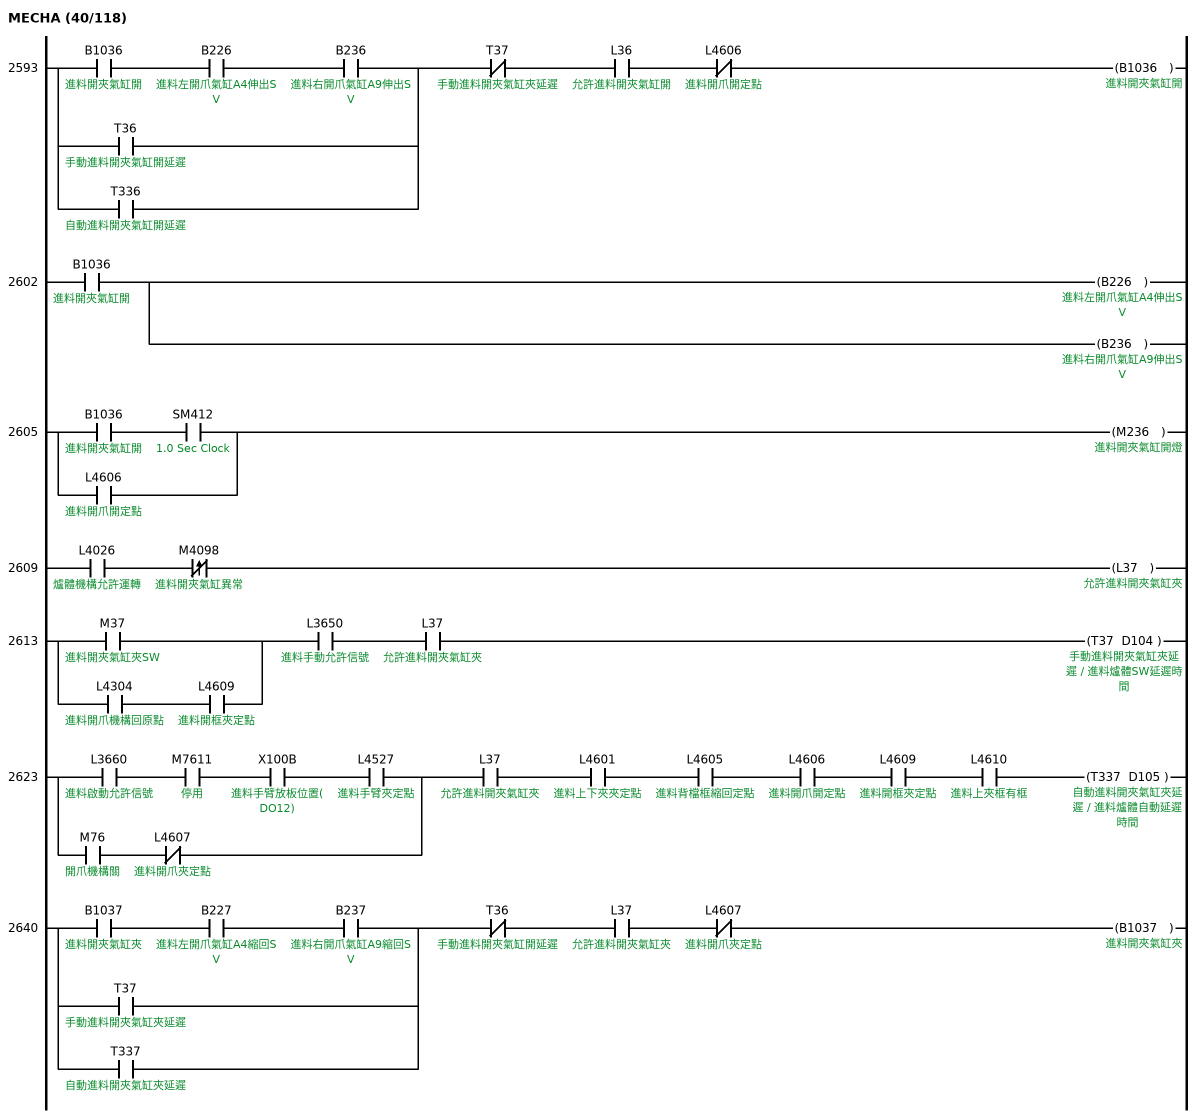
[picture p336: ladder of MECHA, rungs at steps 2593 to 2640]
2593  LD      B1036  ; 進料開夾氣缸開
      AND     B226  ; 進料左開爪氣缸A4伸出SV
      AND     B236  ; 進料右開爪氣缸A9伸出SV
      OR      T36  ; 手動進料開夾氣缸開延遲
      OR      T336  ; 自動進料開夾氣缸開延遲
      ANI     T37  ; 手動進料開夾氣缸夾延遲
      AND     L36  ; 允許進料開夾氣缸開
      ANI     L4606  ; 進料開爪開定點
      OUT     B1036  ; 進料開夾氣缸開
2602  LD      B1036  ; 進料開夾氣缸開
      OUT     B226  ; 進料左開爪氣缸A4伸出SV
      OUT     B236  ; 進料右開爪氣缸A9伸出SV
2605  LD      B1036  ; 進料開夾氣缸開
      AND     SM412  ; 1.0 Sec Clock
      OR      L4606  ; 進料開爪開定點
      OUT     M236  ; 進料開夾氣缸開燈
2609  LD      L4026  ; 爐體機構允許運轉
      ANDPI   M4098  ; 進料開夾氣缸異常
      OUT     L37  ; 允許進料開夾氣缸夾
2613  LD      M37  ; 進料開夾氣缸夾SW
      LD      L4304  ; 進料開爪機構回原點
      AND     L4609  ; 進料開框夾定點
      ORB
      AND     L3650  ; 進料手動允許信號
      AND     L37  ; 允許進料開夾氣缸夾
      OUT     T37 D104  ; 手動進料開夾氣缸夾延遲 / 進料爐體SW延遲時間
2623  LD      L3660  ; 進料啟動允許信號
      AND     M7611  ; 停用
      AND     X100B  ; 進料手臂放板位置(DO12)
      AND     L4527  ; 進料手臂夾定點
      LD      M76  ; 開爪機構關
      ANI     L4607  ; 進料開爪夾定點
      ORB
      AND     L37  ; 允許進料開夾氣缸夾
      AND     L4601  ; 進料上下夾夾定點
      AND     L4605  ; 進料背檔框縮回定點
      AND     L4606  ; 進料開爪開定點
      AND     L4609  ; 進料開框夾定點
      AND     L4610  ; 進料上夾框有框
      OUT     T337 D105  ; 自動進料開夾氣缸夾延遲 / 進料爐體自動延遲時間
2640  LD      B1037  ; 進料開夾氣缸夾
      AND     B227  ; 進料左開爪氣缸A4縮回SV
      AND     B237  ; 進料右開爪氣缸A9縮回SV
      OR      T37  ; 手動進料開夾氣缸夾延遲
      OR      T337  ; 自動進料開夾氣缸夾延遲
      ANI     T36  ; 手動進料開夾氣缸開延遲
      AND     L37  ; 允許進料開夾氣缸夾
      ANI     L4607  ; 進料開爪夾定點
      OUT     B1037  ; 進料開夾氣缸夾
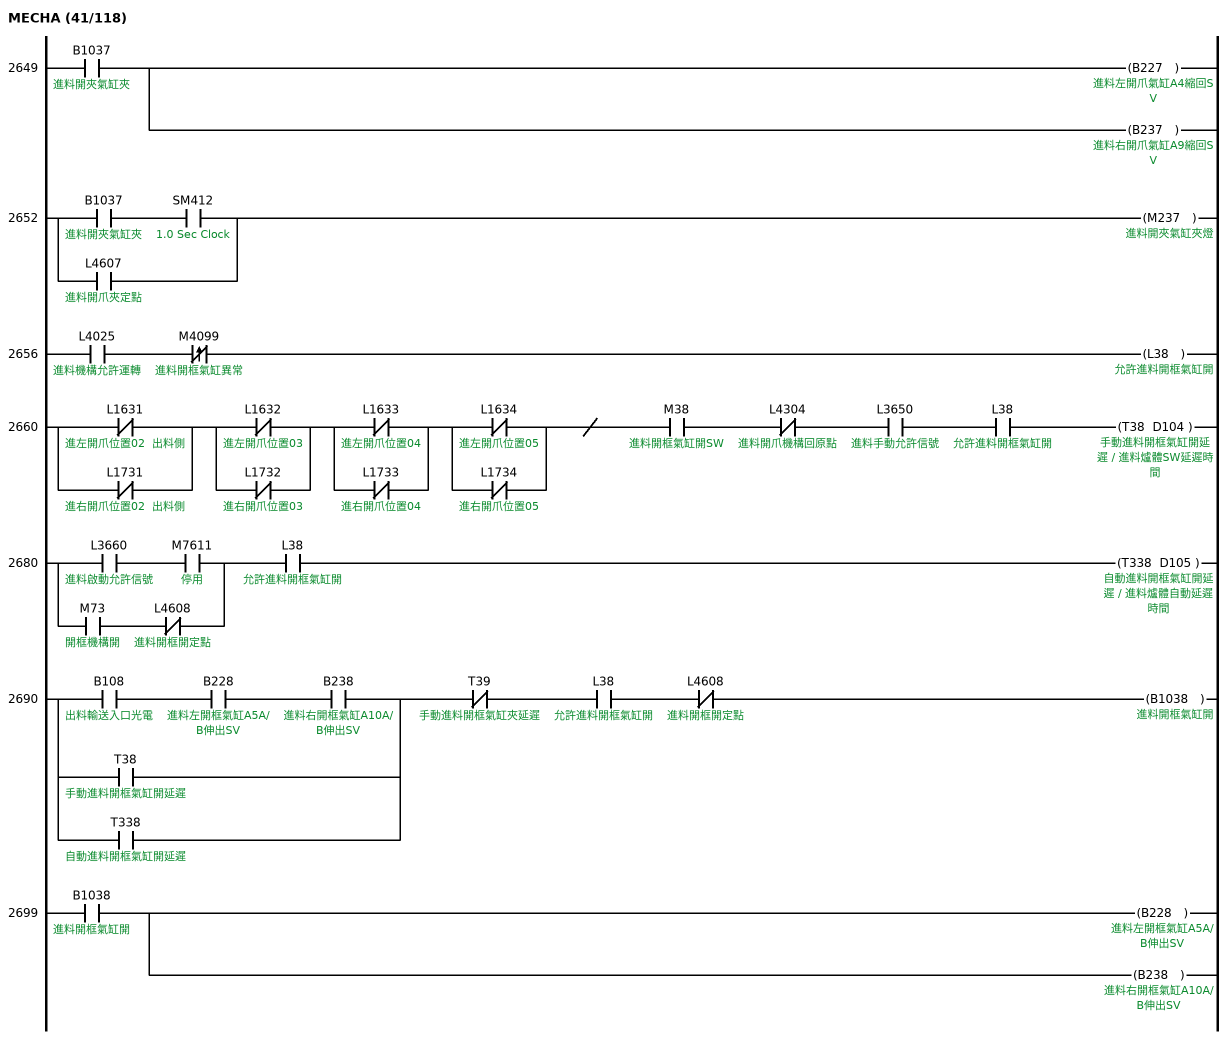
2649  LD      B1037  ; 進料開夾氣缸夾
      OUT     B227  ; 進料左開爪氣缸A4縮回SV
      OUT     B237  ; 進料右開爪氣缸A9縮回SV
2652  LD      B1037  ; 進料開夾氣缸夾
      AND     SM412  ; 1.0 Sec Clock
      OR      L4607  ; 進料開爪夾定點
      OUT     M237  ; 進料開夾氣缸夾燈
2656  LD      L4025  ; 進料機構允許運轉
      ANDPI   M4099  ; 進料開框氣缸異常
      OUT     L38  ; 允許進料開框氣缸開
2660  LDI     L1631  ; 進左開爪位置02  出料側
      ORI     L1731  ; 進右開爪位置02  出料側
      LDI     L1632  ; 進左開爪位置03
      ORI     L1732  ; 進右開爪位置03
      ANB
      LDI     L1633  ; 進左開爪位置04
      ORI     L1733  ; 進右開爪位置04
      ANB
      LDI     L1634  ; 進左開爪位置05
      ORI     L1734  ; 進右開爪位置05
      ANB
      INV
      AND     M38  ; 進料開框氣缸開SW
      ANI     L4304  ; 進料開爪機構回原點
      AND     L3650  ; 進料手動允許信號
      AND     L38  ; 允許進料開框氣缸開
      OUT     T38 D104  ; 手動進料開框氣缸開延遲 / 進料爐體SW延遲時間
2680  LD      L3660  ; 進料啟動允許信號
      AND     M7611  ; 停用
      LD      M73  ; 開框機構開
      ANI     L4608  ; 進料開框開定點
      ORB
      AND     L38  ; 允許進料開框氣缸開
      OUT     T338 D105  ; 自動進料開框氣缸開延遲 / 進料爐體自動延遲時間
2690  LD      B108  ; 出料輸送入口光電
      AND     B228  ; 進料左開框氣缸A5A/B伸出SV
      AND     B238  ; 進料右開框氣缸A10A/B伸出SV
      OR      T38  ; 手動進料開框氣缸開延遲
      OR      T338  ; 自動進料開框氣缸開延遲
      ANI     T39  ; 手動進料開框氣缸夾延遲
      AND     L38  ; 允許進料開框氣缸開
      ANI     L4608  ; 進料開框開定點
      OUT     B1038  ; 進料開框氣缸開
2699  LD      B1038  ; 進料開框氣缸開
      OUT     B228  ; 進料左開框氣缸A5A/B伸出SV
      OUT     B238  ; 進料右開框氣缸A10A/B伸出SV
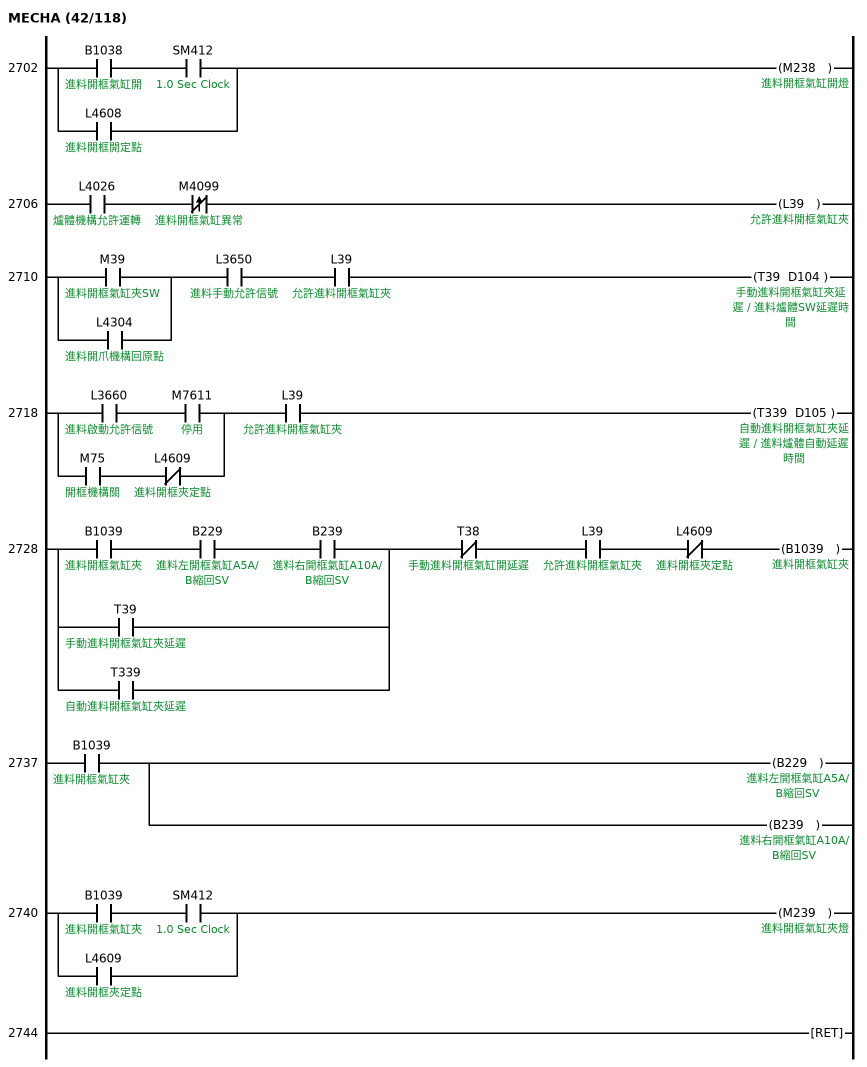
2702  LD      B1038  ; 進料開框氣缸開
      AND     SM412  ; 1.0 Sec Clock
      OR      L4608  ; 進料開框開定點
      OUT     M238  ; 進料開框氣缸開燈
2706  LD      L4026  ; 爐體機構允許運轉
      ANDPI   M4099  ; 進料開框氣缸異常
      OUT     L39  ; 允許進料開框氣缸夾
2710  LD      M39  ; 進料開框氣缸夾SW
      OR      L4304  ; 進料開爪機構回原點
      AND     L3650  ; 進料手動允許信號
      AND     L39  ; 允許進料開框氣缸夾
      OUT     T39 D104  ; 手動進料開框氣缸夾延遲 / 進料爐體SW延遲時間
2718  LD      L3660  ; 進料啟動允許信號
      AND     M7611  ; 停用
      LD      M75  ; 開框機構關
      ANI     L4609  ; 進料開框夾定點
      ORB
      AND     L39  ; 允許進料開框氣缸夾
      OUT     T339 D105  ; 自動進料開框氣缸夾延遲 / 進料爐體自動延遲時間
2728  LD      B1039  ; 進料開框氣缸夾
      AND     B229  ; 進料左開框氣缸A5A/B縮回SV
      AND     B239  ; 進料右開框氣缸A10A/B縮回SV
      OR      T39  ; 手動進料開框氣缸夾延遲
      OR      T339  ; 自動進料開框氣缸夾延遲
      ANI     T38  ; 手動進料開框氣缸開延遲
      AND     L39  ; 允許進料開框氣缸夾
      ANI     L4609  ; 進料開框夾定點
      OUT     B1039  ; 進料開框氣缸夾
2737  LD      B1039  ; 進料開框氣缸夾
      OUT     B229  ; 進料左開框氣缸A5A/B縮回SV
      OUT     B239  ; 進料右開框氣缸A10A/B縮回SV
2740  LD      B1039  ; 進料開框氣缸夾
      AND     SM412  ; 1.0 Sec Clock
      OR      L4609  ; 進料開框夾定點
      OUT     M239  ; 進料開框氣缸夾燈
2744  RET
      P1021
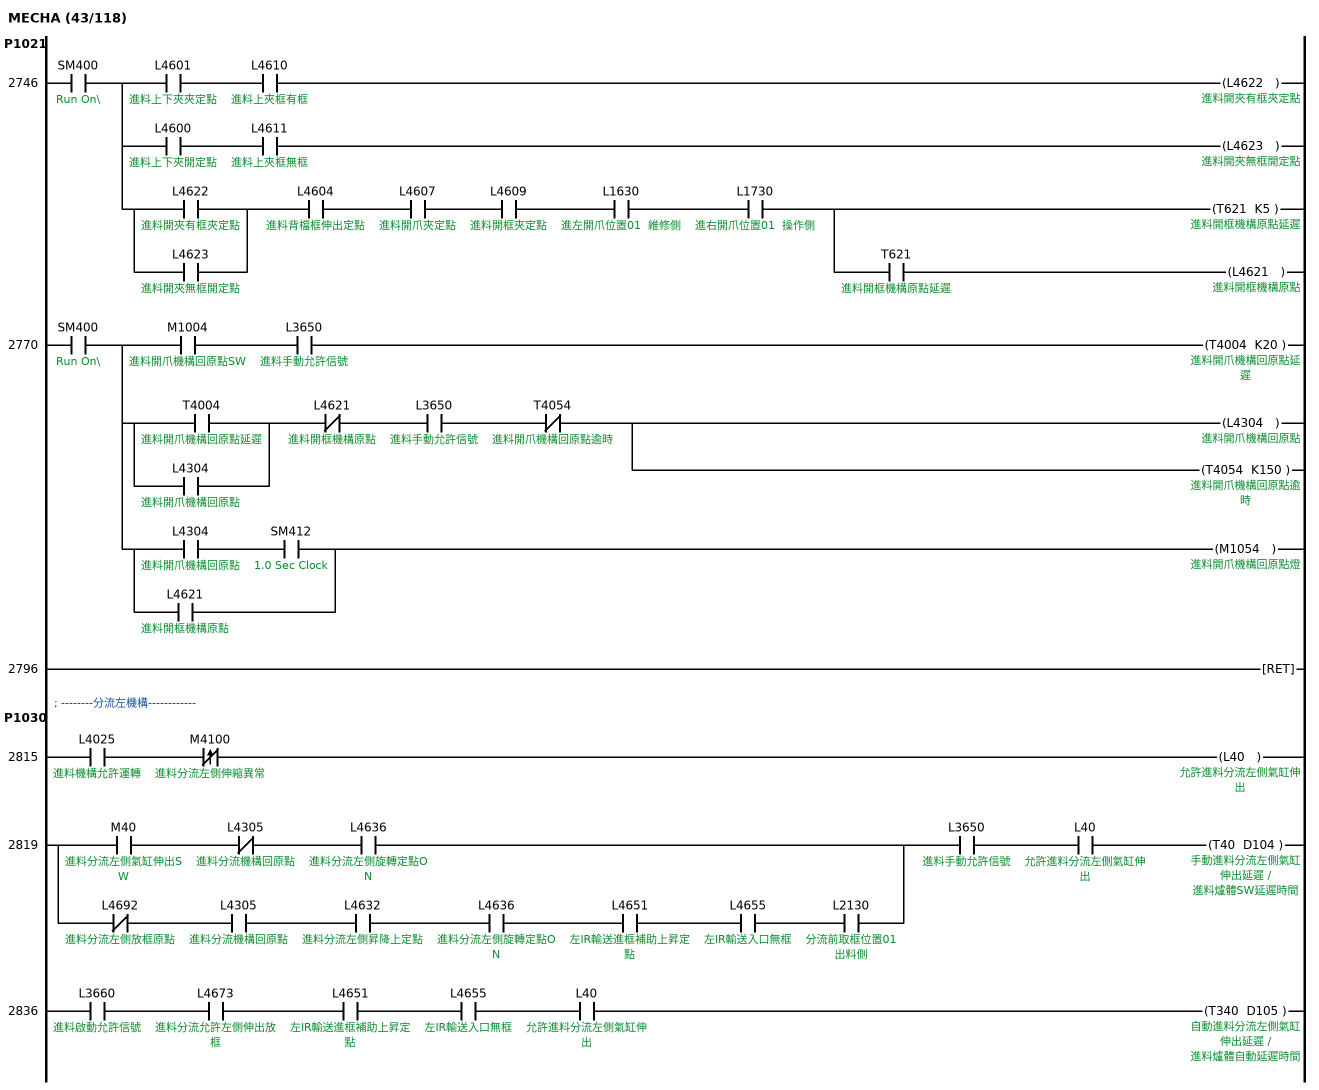
2746  LD      SM400  ; Run On\
      MPS
      AND     L4601  ; 進料上下夾夾定點
      AND     L4610  ; 進料上夾框有框
      OUT     L4622  ; 進料開夾有框夾定點
      MRD
      AND     L4600  ; 進料上下夾開定點
      AND     L4611  ; 進料上夾框無框
      OUT     L4623  ; 進料開夾無框開定點
      MPP
      LD      L4622  ; 進料開夾有框夾定點
      OR      L4623  ; 進料開夾無框開定點
      ANB
      AND     L4604  ; 進料背檔框伸出定點
      AND     L4607  ; 進料開爪夾定點
      AND     L4609  ; 進料開框夾定點
      AND     L1630  ; 進左開爪位置01  維修側
      AND     L1730  ; 進右開爪位置01  操作側
      OUT     T621 K5  ; 進料開框機構原點延遲
      AND     T621  ; 進料開框機構原點延遲
      OUT     L4621  ; 進料開框機構原點
2770  LD      SM400  ; Run On\
      MPS
      AND     M1004  ; 進料開爪機構回原點SW
      AND     L3650  ; 進料手動允許信號
      OUT     T4004 K20  ; 進料開爪機構回原點延遲
      MRD
      LD      T4004  ; 進料開爪機構回原點延遲
      OR      L4304  ; 進料開爪機構回原點
      ANB
      ANI     L4621  ; 進料開框機構原點
      AND     L3650  ; 進料手動允許信號
      ANI     T4054  ; 進料開爪機構回原點逾時
      OUT     L4304  ; 進料開爪機構回原點
      OUT     T4054 K150  ; 進料開爪機構回原點逾時
      MPP
      LD      L4304  ; 進料開爪機構回原點
      AND     SM412  ; 1.0 Sec Clock
      OR      L4621  ; 進料開框機構原點
      ANB
      OUT     M1054  ; 進料開爪機構回原點燈
2796  RET
; --------分流左機構------------
      P1030
2815  LD      L4025  ; 進料機構允許運轉
      ANDPI   M4100  ; 進料分流左側伸縮異常
      OUT     L40  ; 允許進料分流左側氣缸伸出
2819  LD      M40  ; 進料分流左側氣缸伸出SW
      ANI     L4305  ; 進料分流機構回原點
      AND     L4636  ; 進料分流左側旋轉定點ON
      LDI     L4692  ; 進料分流左側放框原點
      AND     L4305  ; 進料分流機構回原點
      AND     L4632  ; 進料分流左側昇降上定點
      AND     L4636  ; 進料分流左側旋轉定點ON
      AND     L4651  ; 左IR輸送進框補助上昇定點
      AND     L4655  ; 左IR輸送入口無框
      AND     L2130  ; 分流前取框位置01  出料側
      ORB
      AND     L3650  ; 進料手動允許信號
      AND     L40  ; 允許進料分流左側氣缸伸出
      OUT     T40 D104  ; 手動進料分流左側氣缸伸出延遲 / 進料爐體SW延遲時間
2836  LD      L3660  ; 進料啟動允許信號
      AND     L4673  ; 進料分流允許左側伸出放框
      AND     L4651  ; 左IR輸送進框補助上昇定點
      AND     L4655  ; 左IR輸送入口無框
      AND     L40  ; 允許進料分流左側氣缸伸出
      OUT     T340 D105  ; 自動進料分流左側氣缸伸出延遲 / 進料爐體自動延遲時間
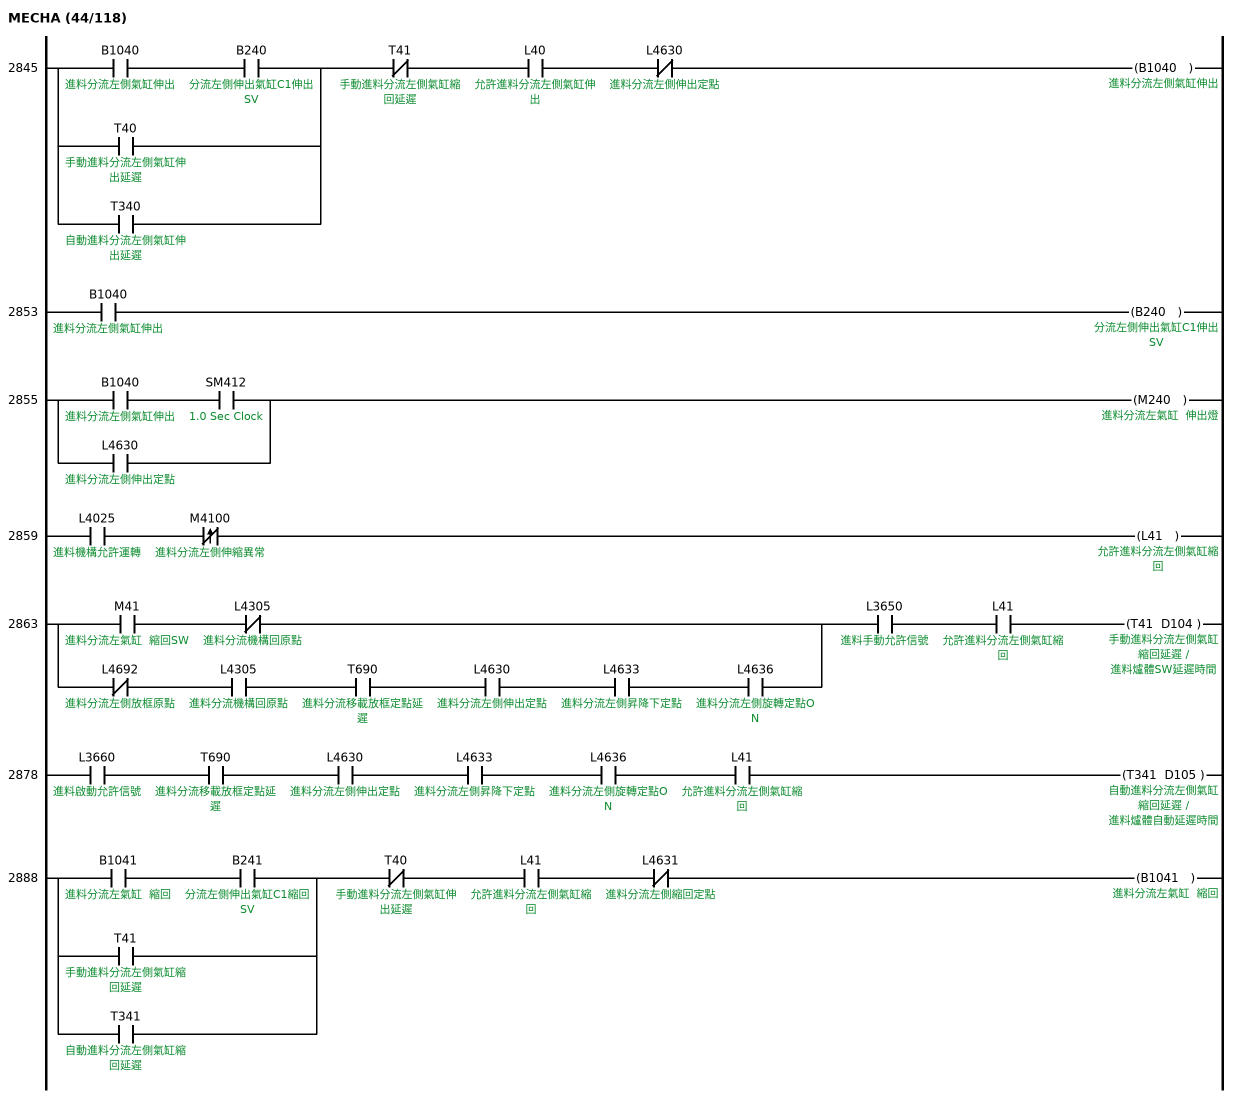
2845  LD      B1040  ; 進料分流左側氣缸伸出
      AND     B240  ; 分流左側伸出氣缸C1伸出SV
      OR      T40  ; 手動進料分流左側氣缸伸出延遲
      OR      T340  ; 自動進料分流左側氣缸伸出延遲
      ANI     T41  ; 手動進料分流左側氣缸縮回延遲
      AND     L40  ; 允許進料分流左側氣缸伸出
      ANI     L4630  ; 進料分流左側伸出定點
      OUT     B1040  ; 進料分流左側氣缸伸出
2853  LD      B1040  ; 進料分流左側氣缸伸出
      OUT     B240  ; 分流左側伸出氣缸C1伸出SV
2855  LD      B1040  ; 進料分流左側氣缸伸出
      AND     SM412  ; 1.0 Sec Clock
      OR      L4630  ; 進料分流左側伸出定點
      OUT     M240  ; 進料分流左氣缸  伸出燈
2859  LD      L4025  ; 進料機構允許運轉
      ANDPI   M4100  ; 進料分流左側伸縮異常
      OUT     L41  ; 允許進料分流左側氣缸縮回
2863  LD      M41  ; 進料分流左氣缸  縮回SW
      ANI     L4305  ; 進料分流機構回原點
      LDI     L4692  ; 進料分流左側放框原點
      AND     L4305  ; 進料分流機構回原點
      AND     T690  ; 進料分流移載放框定點延遲
      AND     L4630  ; 進料分流左側伸出定點
      AND     L4633  ; 進料分流左側昇降下定點
      AND     L4636  ; 進料分流左側旋轉定點ON
      ORB
      AND     L3650  ; 進料手動允許信號
      AND     L41  ; 允許進料分流左側氣缸縮回
      OUT     T41 D104  ; 手動進料分流左側氣缸縮回延遲 / 進料爐體SW延遲時間
2878  LD      L3660  ; 進料啟動允許信號
      AND     T690  ; 進料分流移載放框定點延遲
      AND     L4630  ; 進料分流左側伸出定點
      AND     L4633  ; 進料分流左側昇降下定點
      AND     L4636  ; 進料分流左側旋轉定點ON
      AND     L41  ; 允許進料分流左側氣缸縮回
      OUT     T341 D105  ; 自動進料分流左側氣缸縮回延遲 / 進料爐體自動延遲時間
2888  LD      B1041  ; 進料分流左氣缸  縮回
      AND     B241  ; 分流左側伸出氣缸C1縮回SV
      OR      T41  ; 手動進料分流左側氣缸縮回延遲
      OR      T341  ; 自動進料分流左側氣缸縮回延遲
      ANI     T40  ; 手動進料分流左側氣缸伸出延遲
      AND     L41  ; 允許進料分流左側氣缸縮回
      ANI     L4631  ; 進料分流左側縮回定點
      OUT     B1041  ; 進料分流左氣缸  縮回
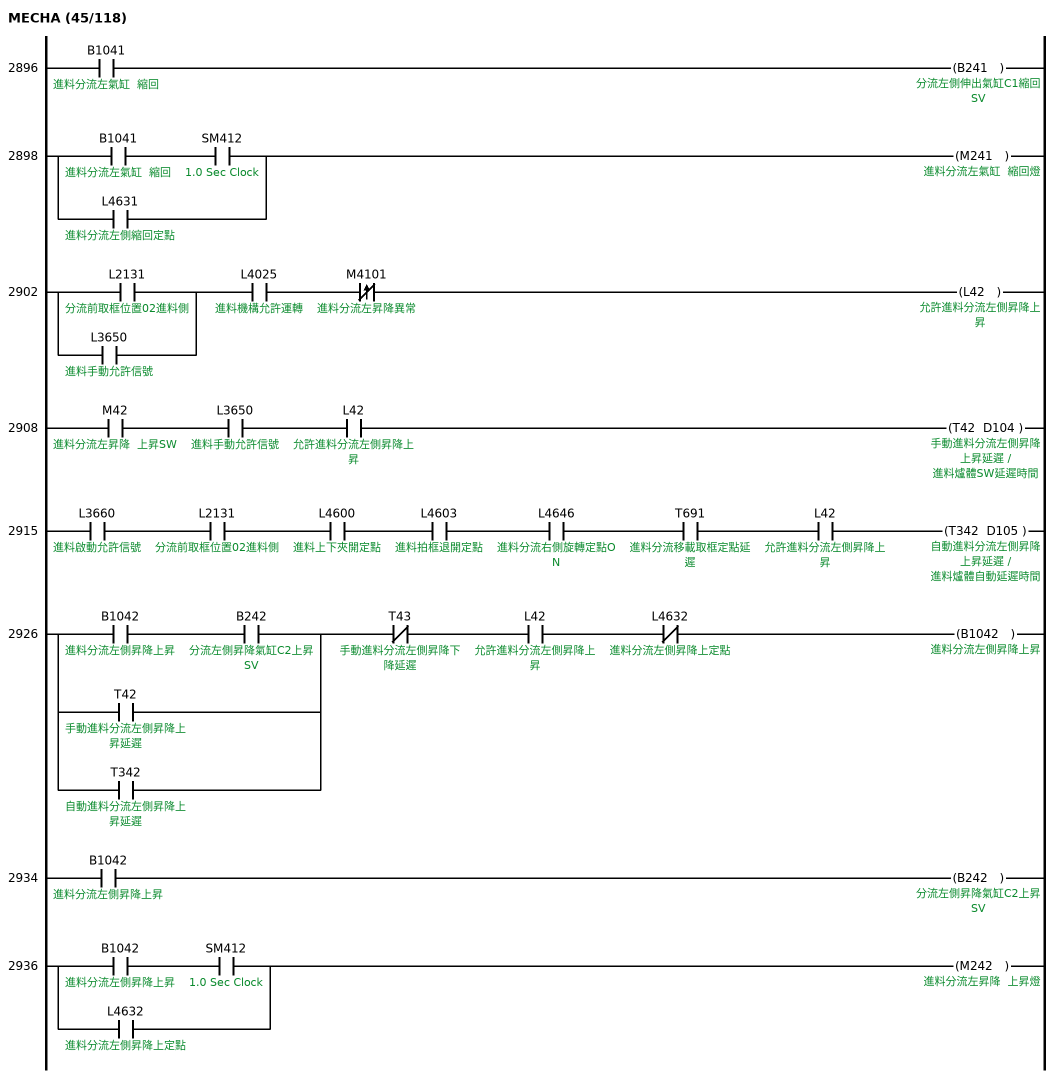
2896  LD      B1041  ; 進料分流左氣缸  縮回
      OUT     B241  ; 分流左側伸出氣缸C1縮回SV
2898  LD      B1041  ; 進料分流左氣缸  縮回
      AND     SM412  ; 1.0 Sec Clock
      OR      L4631  ; 進料分流左側縮回定點
      OUT     M241  ; 進料分流左氣缸  縮回燈
2902  LD      L2131  ; 分流前取框位置02進料側
      OR      L3650  ; 進料手動允許信號
      AND     L4025  ; 進料機構允許運轉
      ANDPI   M4101  ; 進料分流左昇降異常
      OUT     L42  ; 允許進料分流左側昇降上昇
2908  LD      M42  ; 進料分流左昇降  上昇SW
      AND     L3650  ; 進料手動允許信號
      AND     L42  ; 允許進料分流左側昇降上昇
      OUT     T42 D104  ; 手動進料分流左側昇降上昇延遲 / 進料爐體SW延遲時間
2915  LD      L3660  ; 進料啟動允許信號
      AND     L2131  ; 分流前取框位置02進料側
      AND     L4600  ; 進料上下夾開定點
      AND     L4603  ; 進料拍框退開定點
      AND     L4646  ; 進料分流右側旋轉定點ON
      AND     T691  ; 進料分流移載取框定點延遲
      AND     L42  ; 允許進料分流左側昇降上昇
      OUT     T342 D105  ; 自動進料分流左側昇降上昇延遲 / 進料爐體自動延遲時間
2926  LD      B1042  ; 進料分流左側昇降上昇
      AND     B242  ; 分流左側昇降氣缸C2上昇SV
      OR      T42  ; 手動進料分流左側昇降上昇延遲
      OR      T342  ; 自動進料分流左側昇降上昇延遲
      ANI     T43  ; 手動進料分流左側昇降下降延遲
      AND     L42  ; 允許進料分流左側昇降上昇
      ANI     L4632  ; 進料分流左側昇降上定點
      OUT     B1042  ; 進料分流左側昇降上昇
2934  LD      B1042  ; 進料分流左側昇降上昇
      OUT     B242  ; 分流左側昇降氣缸C2上昇SV
2936  LD      B1042  ; 進料分流左側昇降上昇
      AND     SM412  ; 1.0 Sec Clock
      OR      L4632  ; 進料分流左側昇降上定點
      OUT     M242  ; 進料分流左昇降  上昇燈
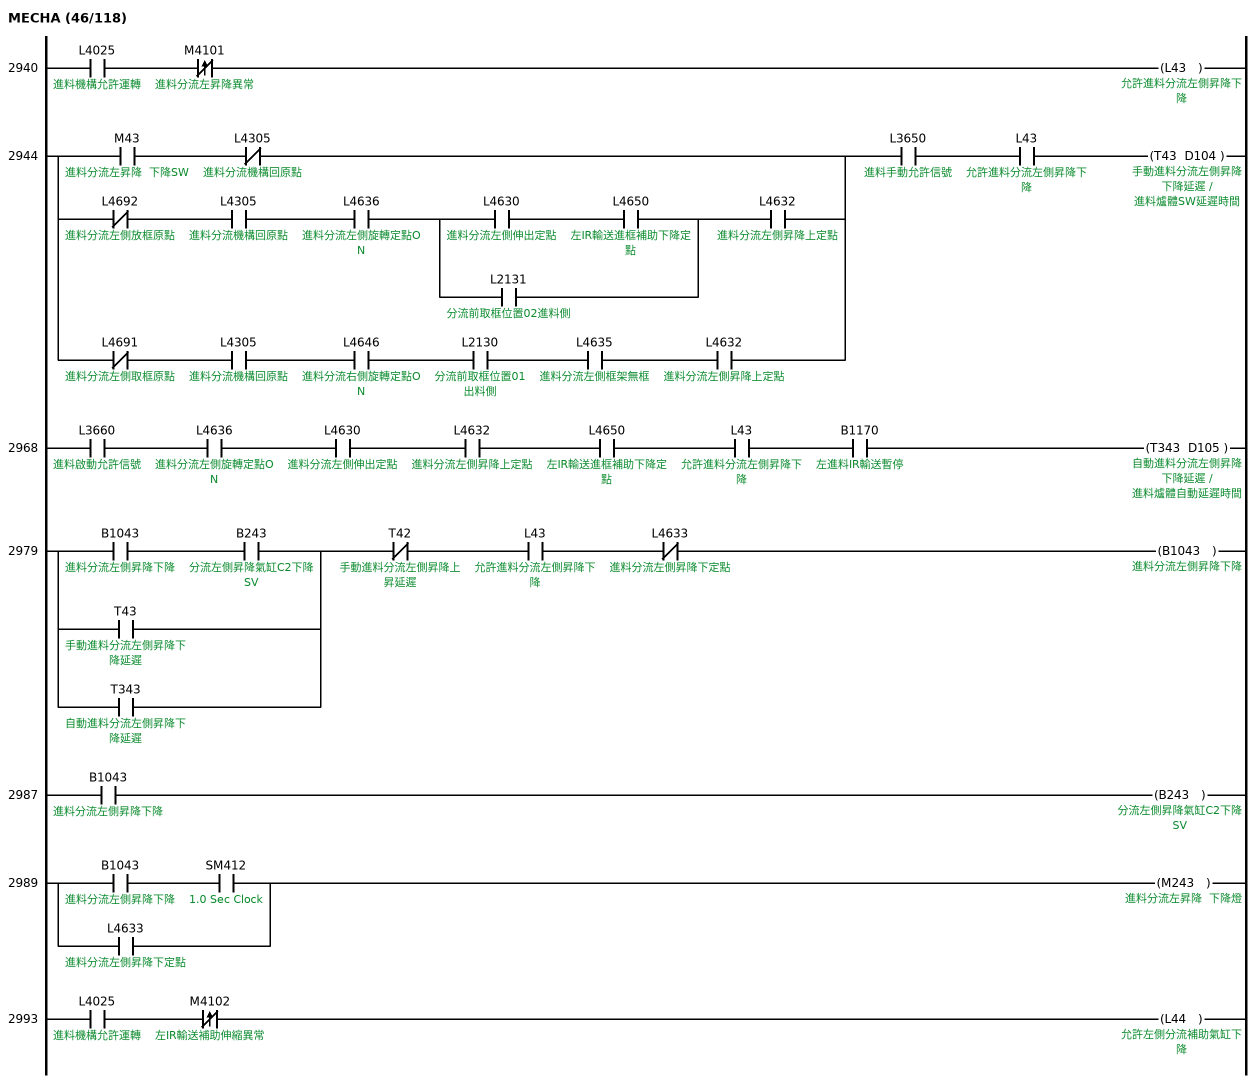
2940  LD      L4025  ; 進料機構允許運轉
      ANDPI   M4101  ; 進料分流左昇降異常
      OUT     L43  ; 允許進料分流左側昇降下降
2944  LD      M43  ; 進料分流左昇降  下降SW
      ANI     L4305  ; 進料分流機構回原點
      LDI     L4692  ; 進料分流左側放框原點
      AND     L4305  ; 進料分流機構回原點
      AND     L4636  ; 進料分流左側旋轉定點ON
      LD      L4630  ; 進料分流左側伸出定點
      AND     L4650  ; 左IR輸送進框補助下降定點
      OR      L2131  ; 分流前取框位置02進料側
      ANB
      AND     L4632  ; 進料分流左側昇降上定點
      ORB
      LDI     L4691  ; 進料分流左側取框原點
      AND     L4305  ; 進料分流機構回原點
      AND     L4646  ; 進料分流右側旋轉定點ON
      AND     L2130  ; 分流前取框位置01  出料側
      AND     L4635  ; 進料分流左側框架無框
      AND     L4632  ; 進料分流左側昇降上定點
      ORB
      AND     L3650  ; 進料手動允許信號
      AND     L43  ; 允許進料分流左側昇降下降
      OUT     T43 D104  ; 手動進料分流左側昇降下降延遲 / 進料爐體SW延遲時間
2968  LD      L3660  ; 進料啟動允許信號
      AND     L4636  ; 進料分流左側旋轉定點ON
      AND     L4630  ; 進料分流左側伸出定點
      AND     L4632  ; 進料分流左側昇降上定點
      AND     L4650  ; 左IR輸送進框補助下降定點
      AND     L43  ; 允許進料分流左側昇降下降
      AND     B1170  ; 左進料IR輸送暫停
      OUT     T343 D105  ; 自動進料分流左側昇降下降延遲 / 進料爐體自動延遲時間
2979  LD      B1043  ; 進料分流左側昇降下降
      AND     B243  ; 分流左側昇降氣缸C2下降SV
      OR      T43  ; 手動進料分流左側昇降下降延遲
      OR      T343  ; 自動進料分流左側昇降下降延遲
      ANI     T42  ; 手動進料分流左側昇降上昇延遲
      AND     L43  ; 允許進料分流左側昇降下降
      ANI     L4633  ; 進料分流左側昇降下定點
      OUT     B1043  ; 進料分流左側昇降下降
2987  LD      B1043  ; 進料分流左側昇降下降
      OUT     B243  ; 分流左側昇降氣缸C2下降SV
2989  LD      B1043  ; 進料分流左側昇降下降
      AND     SM412  ; 1.0 Sec Clock
      OR      L4633  ; 進料分流左側昇降下定點
      OUT     M243  ; 進料分流左昇降  下降燈
2993  LD      L4025  ; 進料機構允許運轉
      ANDPI   M4102  ; 左IR輸送補助伸縮異常
      OUT     L44  ; 允許左側分流補助氣缸下降
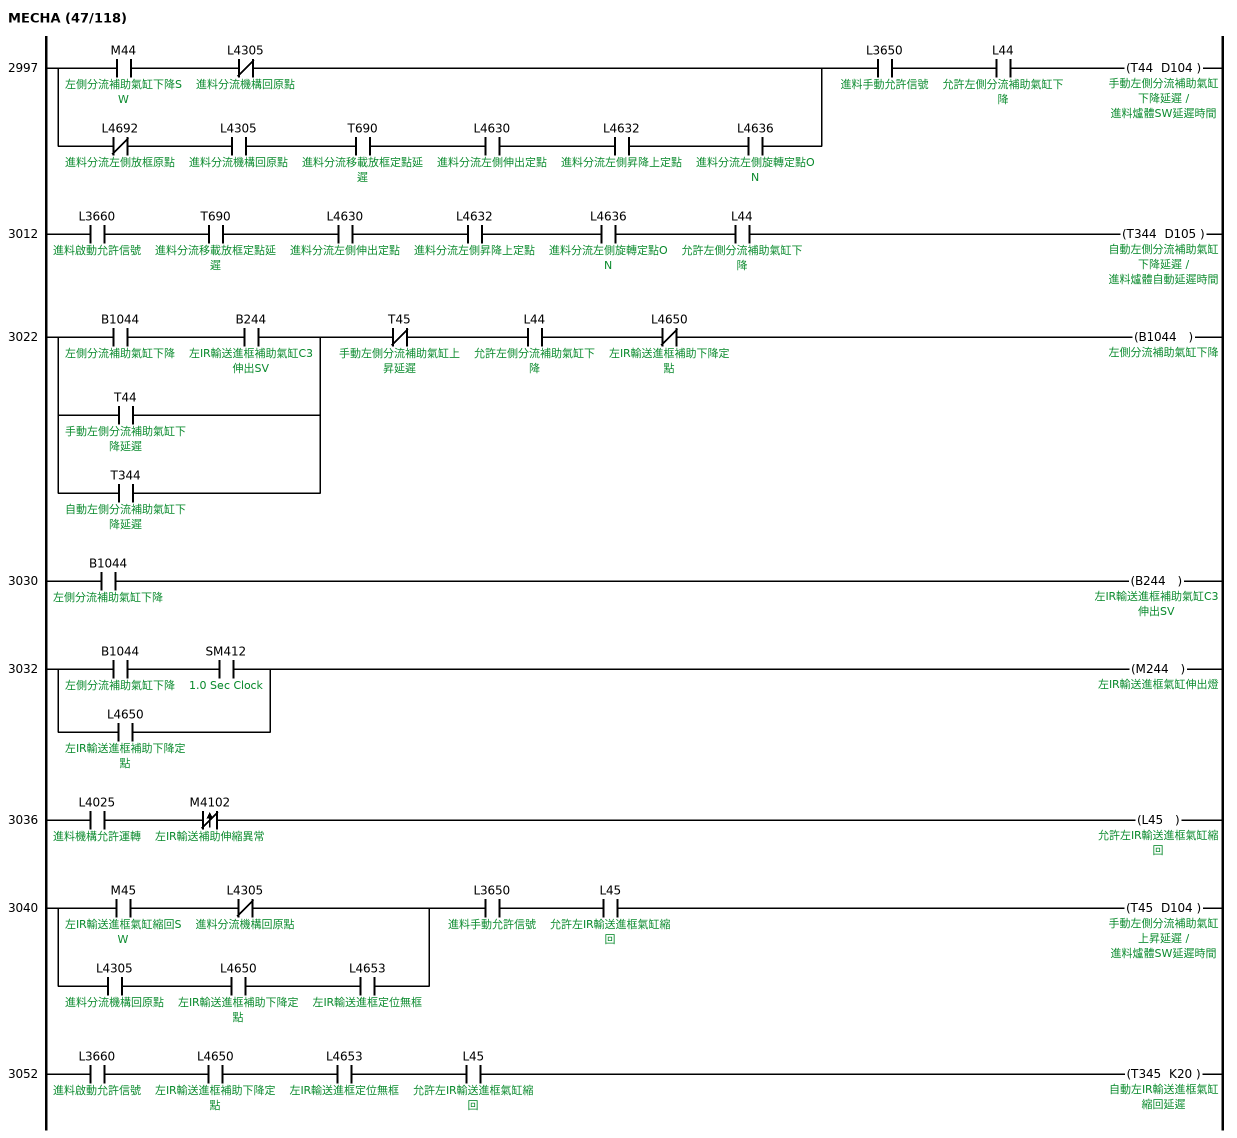
2997  LD      M44  ; 左側分流補助氣缸下降SW
      ANI     L4305  ; 進料分流機構回原點
      LDI     L4692  ; 進料分流左側放框原點
      AND     L4305  ; 進料分流機構回原點
      AND     T690  ; 進料分流移載放框定點延遲
      AND     L4630  ; 進料分流左側伸出定點
      AND     L4632  ; 進料分流左側昇降上定點
      AND     L4636  ; 進料分流左側旋轉定點ON
      ORB
      AND     L3650  ; 進料手動允許信號
      AND     L44  ; 允許左側分流補助氣缸下降
      OUT     T44 D104  ; 手動左側分流補助氣缸下降延遲 / 進料爐體SW延遲時間
3012  LD      L3660  ; 進料啟動允許信號
      AND     T690  ; 進料分流移載放框定點延遲
      AND     L4630  ; 進料分流左側伸出定點
      AND     L4632  ; 進料分流左側昇降上定點
      AND     L4636  ; 進料分流左側旋轉定點ON
      AND     L44  ; 允許左側分流補助氣缸下降
      OUT     T344 D105  ; 自動左側分流補助氣缸下降延遲 / 進料爐體自動延遲時間
3022  LD      B1044  ; 左側分流補助氣缸下降
      AND     B244  ; 左IR輸送進框補助氣缸C3伸出SV
      OR      T44  ; 手動左側分流補助氣缸下降延遲
      OR      T344  ; 自動左側分流補助氣缸下降延遲
      ANI     T45  ; 手動左側分流補助氣缸上昇延遲
      AND     L44  ; 允許左側分流補助氣缸下降
      ANI     L4650  ; 左IR輸送進框補助下降定點
      OUT     B1044  ; 左側分流補助氣缸下降
3030  LD      B1044  ; 左側分流補助氣缸下降
      OUT     B244  ; 左IR輸送進框補助氣缸C3伸出SV
3032  LD      B1044  ; 左側分流補助氣缸下降
      AND     SM412  ; 1.0 Sec Clock
      OR      L4650  ; 左IR輸送進框補助下降定點
      OUT     M244  ; 左IR輸送進框氣缸伸出燈
3036  LD      L4025  ; 進料機構允許運轉
      ANDPI   M4102  ; 左IR輸送補助伸縮異常
      OUT     L45  ; 允許左IR輸送進框氣缸縮回
3040  LD      M45  ; 左IR輸送進框氣缸縮回SW
      ANI     L4305  ; 進料分流機構回原點
      LD      L4305  ; 進料分流機構回原點
      AND     L4650  ; 左IR輸送進框補助下降定點
      AND     L4653  ; 左IR輸送進框定位無框
      ORB
      AND     L3650  ; 進料手動允許信號
      AND     L45  ; 允許左IR輸送進框氣缸縮回
      OUT     T45 D104  ; 手動左側分流補助氣缸上昇延遲 / 進料爐體SW延遲時間
3052  LD      L3660  ; 進料啟動允許信號
      AND     L4650  ; 左IR輸送進框補助下降定點
      AND     L4653  ; 左IR輸送進框定位無框
      AND     L45  ; 允許左IR輸送進框氣缸縮回
      OUT     T345 K20  ; 自動左IR輸送進框氣缸縮回延遲
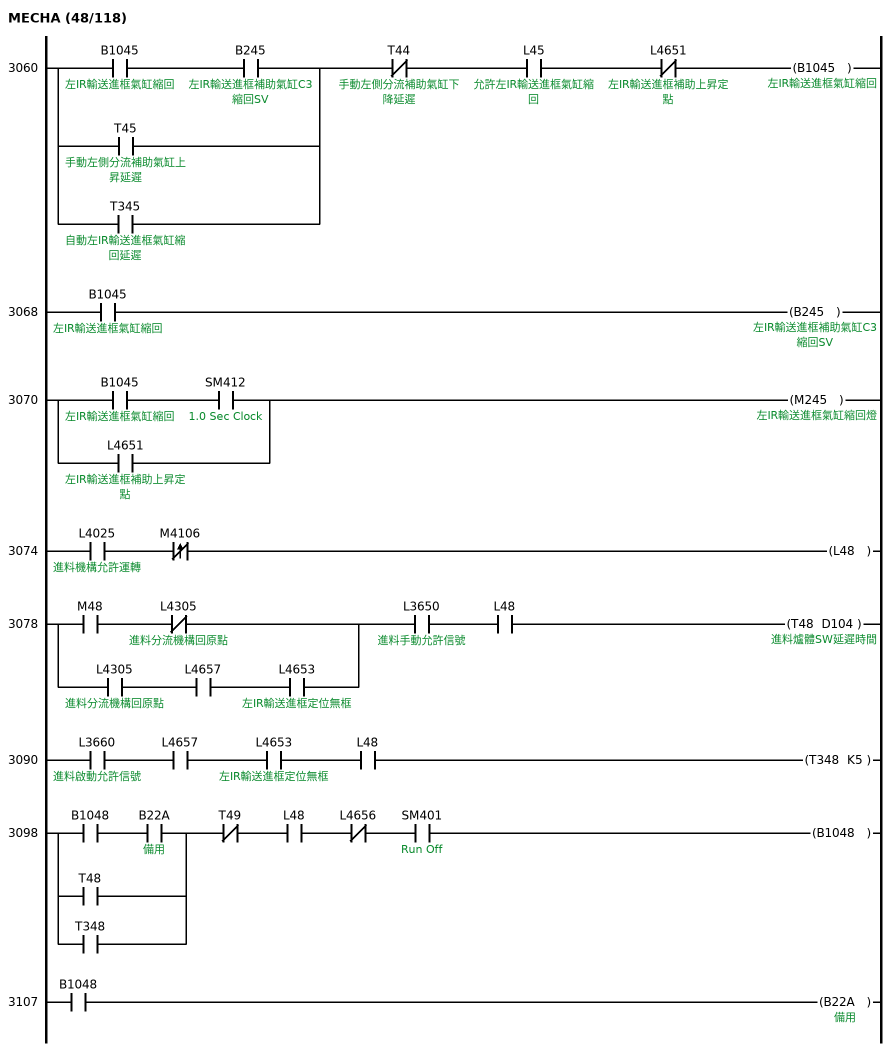
3060  LD      B1045  ; 左IR輸送進框氣缸縮回
      AND     B245  ; 左IR輸送進框補助氣缸C3縮回SV
      OR      T45  ; 手動左側分流補助氣缸上昇延遲
      OR      T345  ; 自動左IR輸送進框氣缸縮回延遲
      ANI     T44  ; 手動左側分流補助氣缸下降延遲
      AND     L45  ; 允許左IR輸送進框氣缸縮回
      ANI     L4651  ; 左IR輸送進框補助上昇定點
      OUT     B1045  ; 左IR輸送進框氣缸縮回
3068  LD      B1045  ; 左IR輸送進框氣缸縮回
      OUT     B245  ; 左IR輸送進框補助氣缸C3縮回SV
3070  LD      B1045  ; 左IR輸送進框氣缸縮回
      AND     SM412  ; 1.0 Sec Clock
      OR      L4651  ; 左IR輸送進框補助上昇定點
      OUT     M245  ; 左IR輸送進框氣缸縮回燈
3074  LD      L4025  ; 進料機構允許運轉
      ANDPI   M4106
      OUT     L48
3078  LD      M48
      ANI     L4305  ; 進料分流機構回原點
      LD      L4305  ; 進料分流機構回原點
      AND     L4657
      AND     L4653  ; 左IR輸送進框定位無框
      ORB
      AND     L3650  ; 進料手動允許信號
      AND     L48
      OUT     T48 D104  ; 進料爐體SW延遲時間
3090  LD      L3660  ; 進料啟動允許信號
      AND     L4657
      AND     L4653  ; 左IR輸送進框定位無框
      AND     L48
      OUT     T348 K5
3098  LD      B1048
      AND     B22A  ; 備用
      OR      T48
      OR      T348
      ANI     T49
      AND     L48
      ANI     L4656
      AND     SM401  ; Run Off
      OUT     B1048
3107  LD      B1048
      OUT     B22A  ; 備用
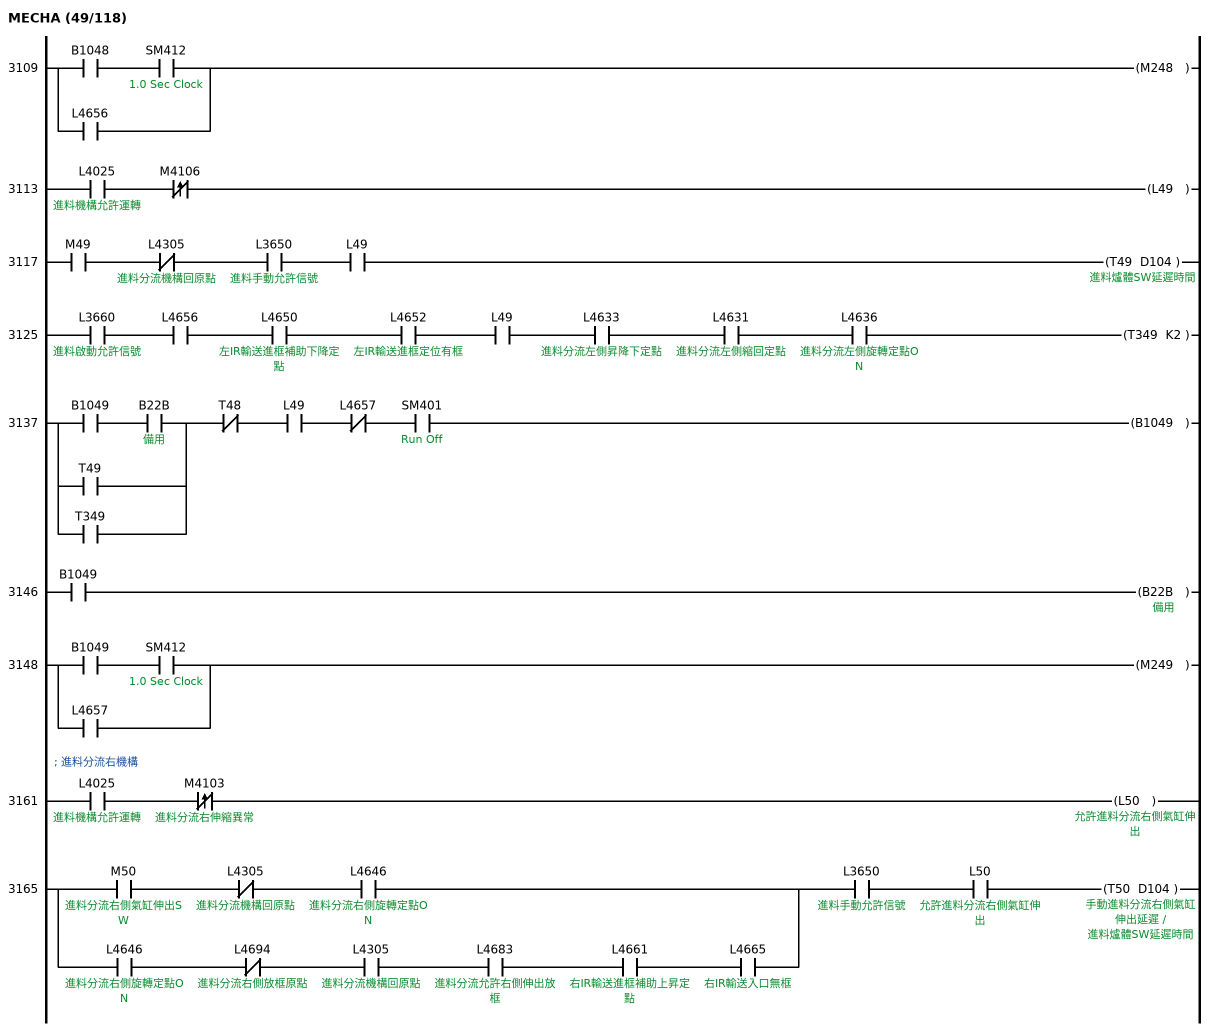
3109  LD      B1048
      AND     SM412  ; 1.0 Sec Clock
      OR      L4656
      OUT     M248
3113  LD      L4025  ; 進料機構允許運轉
      ANDPI   M4106
      OUT     L49
3117  LD      M49
      ANI     L4305  ; 進料分流機構回原點
      AND     L3650  ; 進料手動允許信號
      AND     L49
      OUT     T49 D104  ; 進料爐體SW延遲時間
3125  LD      L3660  ; 進料啟動允許信號
      AND     L4656
      AND     L4650  ; 左IR輸送進框補助下降定點
      AND     L4652  ; 左IR輸送進框定位有框
      AND     L49
      AND     L4633  ; 進料分流左側昇降下定點
      AND     L4631  ; 進料分流左側縮回定點
      AND     L4636  ; 進料分流左側旋轉定點ON
      OUT     T349 K2
3137  LD      B1049
      AND     B22B  ; 備用
      OR      T49
      OR      T349
      ANI     T48
      AND     L49
      ANI     L4657
      AND     SM401  ; Run Off
      OUT     B1049
3146  LD      B1049
      OUT     B22B  ; 備用
3148  LD      B1049
      AND     SM412  ; 1.0 Sec Clock
      OR      L4657
      OUT     M249
; 進料分流右機構
3161  LD      L4025  ; 進料機構允許運轉
      ANDPI   M4103  ; 進料分流右伸縮異常
      OUT     L50  ; 允許進料分流右側氣缸伸出
3165  LD      M50  ; 進料分流右側氣缸伸出SW
      ANI     L4305  ; 進料分流機構回原點
      AND     L4646  ; 進料分流右側旋轉定點ON
      LD      L4646  ; 進料分流右側旋轉定點ON
      ANI     L4694  ; 進料分流右側放框原點
      AND     L4305  ; 進料分流機構回原點
      AND     L4683  ; 進料分流允許右側伸出放框
      AND     L4661  ; 右IR輸送進框補助上昇定點
      AND     L4665  ; 右IR輸送入口無框
      ORB
      AND     L3650  ; 進料手動允許信號
      AND     L50  ; 允許進料分流右側氣缸伸出
      OUT     T50 D104  ; 手動進料分流右側氣缸伸出延遲 / 進料爐體SW延遲時間
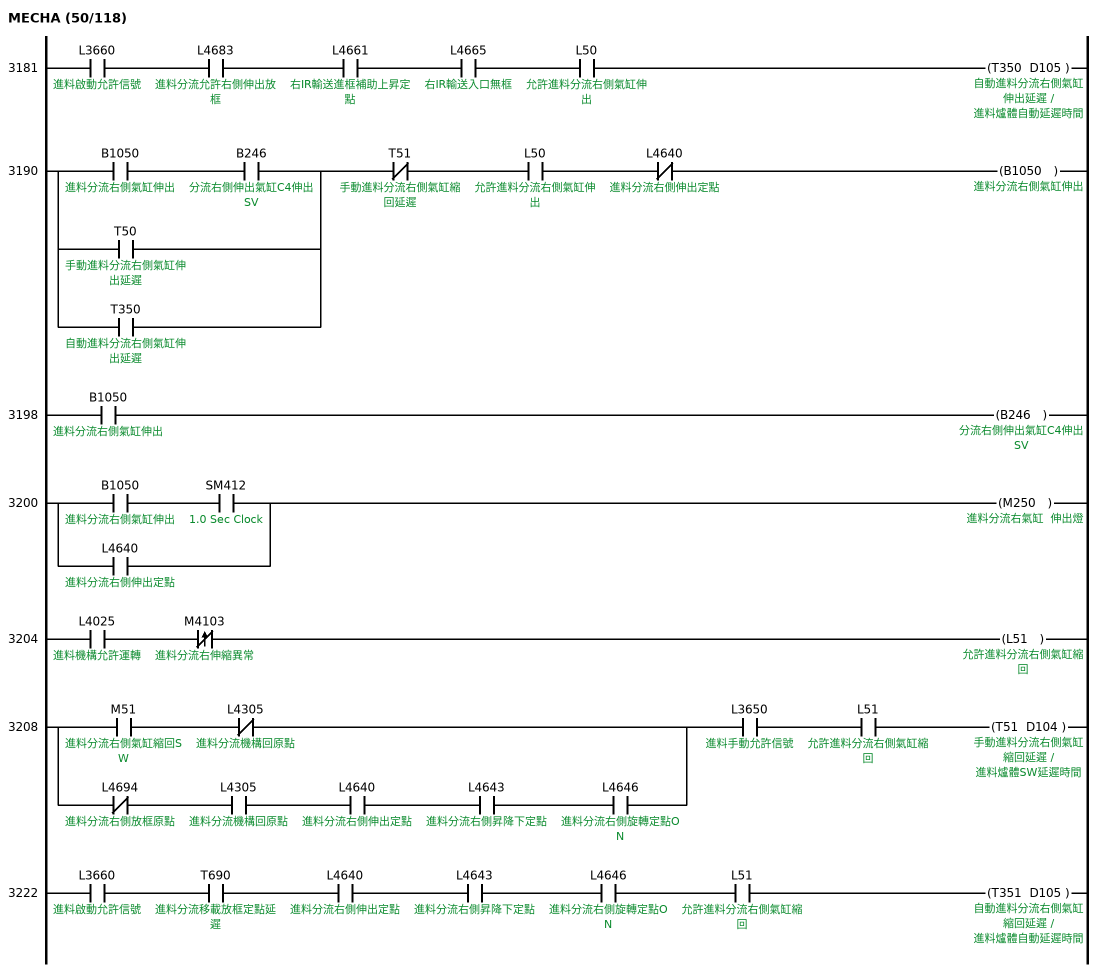
3181  LD      L3660  ; 進料啟動允許信號
      AND     L4683  ; 進料分流允許右側伸出放框
      AND     L4661  ; 右IR輸送進框補助上昇定點
      AND     L4665  ; 右IR輸送入口無框
      AND     L50  ; 允許進料分流右側氣缸伸出
      OUT     T350 D105  ; 自動進料分流右側氣缸伸出延遲 / 進料爐體自動延遲時間
3190  LD      B1050  ; 進料分流右側氣缸伸出
      AND     B246  ; 分流右側伸出氣缸C4伸出SV
      OR      T50  ; 手動進料分流右側氣缸伸出延遲
      OR      T350  ; 自動進料分流右側氣缸伸出延遲
      ANI     T51  ; 手動進料分流右側氣缸縮回延遲
      AND     L50  ; 允許進料分流右側氣缸伸出
      ANI     L4640  ; 進料分流右側伸出定點
      OUT     B1050  ; 進料分流右側氣缸伸出
3198  LD      B1050  ; 進料分流右側氣缸伸出
      OUT     B246  ; 分流右側伸出氣缸C4伸出SV
3200  LD      B1050  ; 進料分流右側氣缸伸出
      AND     SM412  ; 1.0 Sec Clock
      OR      L4640  ; 進料分流右側伸出定點
      OUT     M250  ; 進料分流右氣缸  伸出燈
3204  LD      L4025  ; 進料機構允許運轉
      ANDPI   M4103  ; 進料分流右伸縮異常
      OUT     L51  ; 允許進料分流右側氣缸縮回
3208  LD      M51  ; 進料分流右側氣缸縮回SW
      ANI     L4305  ; 進料分流機構回原點
      LDI     L4694  ; 進料分流右側放框原點
      AND     L4305  ; 進料分流機構回原點
      AND     L4640  ; 進料分流右側伸出定點
      AND     L4643  ; 進料分流右側昇降下定點
      AND     L4646  ; 進料分流右側旋轉定點ON
      ORB
      AND     L3650  ; 進料手動允許信號
      AND     L51  ; 允許進料分流右側氣缸縮回
      OUT     T51 D104  ; 手動進料分流右側氣缸縮回延遲 / 進料爐體SW延遲時間
3222  LD      L3660  ; 進料啟動允許信號
      AND     T690  ; 進料分流移載放框定點延遲
      AND     L4640  ; 進料分流右側伸出定點
      AND     L4643  ; 進料分流右側昇降下定點
      AND     L4646  ; 進料分流右側旋轉定點ON
      AND     L51  ; 允許進料分流右側氣缸縮回
      OUT     T351 D105  ; 自動進料分流右側氣缸縮回延遲 / 進料爐體自動延遲時間
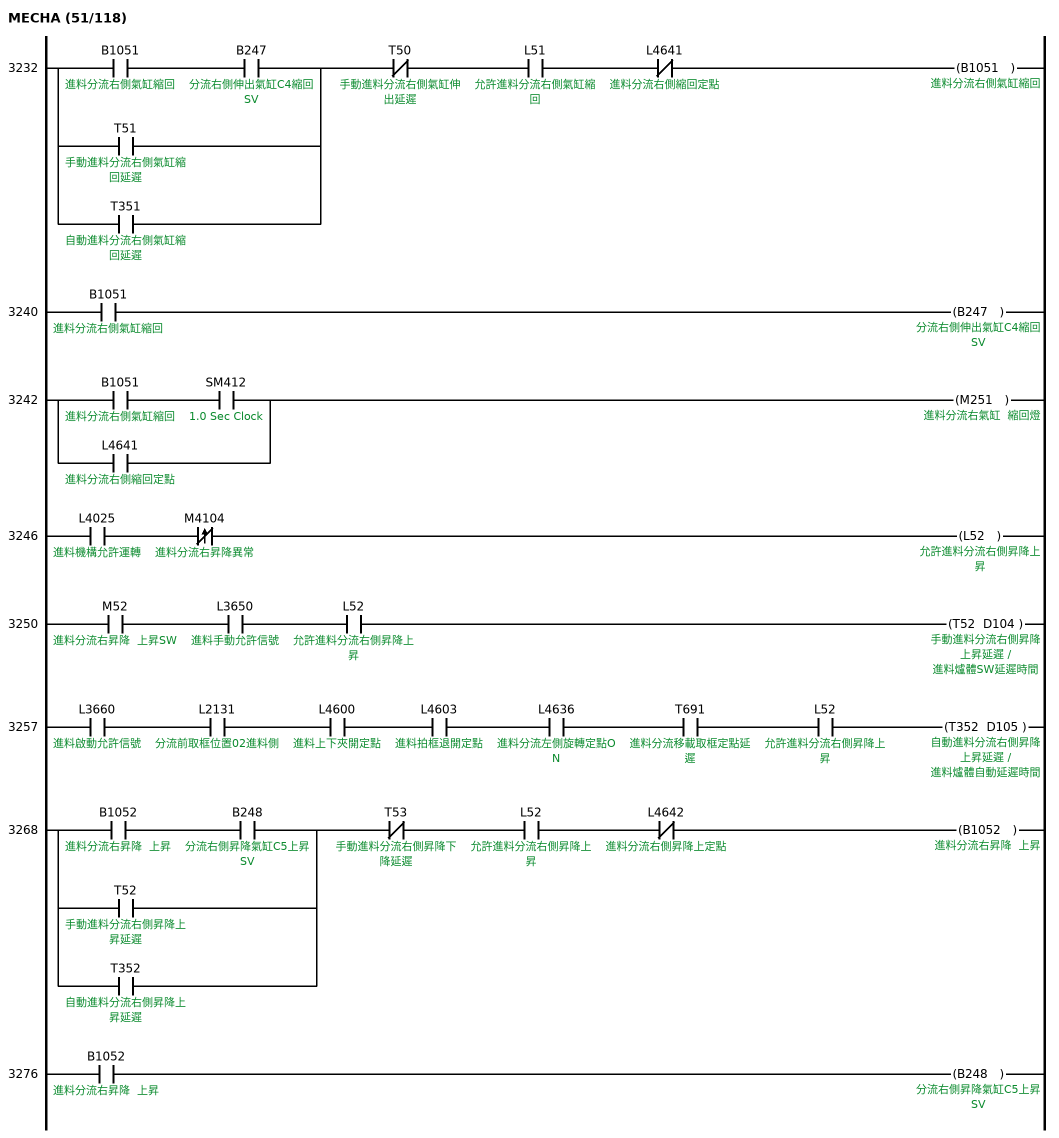
3232  LD      B1051  ; 進料分流右側氣缸縮回
      AND     B247  ; 分流右側伸出氣缸C4縮回SV
      OR      T51  ; 手動進料分流右側氣缸縮回延遲
      OR      T351  ; 自動進料分流右側氣缸縮回延遲
      ANI     T50  ; 手動進料分流右側氣缸伸出延遲
      AND     L51  ; 允許進料分流右側氣缸縮回
      ANI     L4641  ; 進料分流右側縮回定點
      OUT     B1051  ; 進料分流右側氣缸縮回
3240  LD      B1051  ; 進料分流右側氣缸縮回
      OUT     B247  ; 分流右側伸出氣缸C4縮回SV
3242  LD      B1051  ; 進料分流右側氣缸縮回
      AND     SM412  ; 1.0 Sec Clock
      OR      L4641  ; 進料分流右側縮回定點
      OUT     M251  ; 進料分流右氣缸  縮回燈
3246  LD      L4025  ; 進料機構允許運轉
      ANDPI   M4104  ; 進料分流右昇降異常
      OUT     L52  ; 允許進料分流右側昇降上昇
3250  LD      M52  ; 進料分流右昇降  上昇SW
      AND     L3650  ; 進料手動允許信號
      AND     L52  ; 允許進料分流右側昇降上昇
      OUT     T52 D104  ; 手動進料分流右側昇降上昇延遲 / 進料爐體SW延遲時間
3257  LD      L3660  ; 進料啟動允許信號
      AND     L2131  ; 分流前取框位置02進料側
      AND     L4600  ; 進料上下夾開定點
      AND     L4603  ; 進料拍框退開定點
      AND     L4636  ; 進料分流左側旋轉定點ON
      AND     T691  ; 進料分流移載取框定點延遲
      AND     L52  ; 允許進料分流右側昇降上昇
      OUT     T352 D105  ; 自動進料分流右側昇降上昇延遲 / 進料爐體自動延遲時間
3268  LD      B1052  ; 進料分流右昇降  上昇
      AND     B248  ; 分流右側昇降氣缸C5上昇SV
      OR      T52  ; 手動進料分流右側昇降上昇延遲
      OR      T352  ; 自動進料分流右側昇降上昇延遲
      ANI     T53  ; 手動進料分流右側昇降下降延遲
      AND     L52  ; 允許進料分流右側昇降上昇
      ANI     L4642  ; 進料分流右側昇降上定點
      OUT     B1052  ; 進料分流右昇降  上昇
3276  LD      B1052  ; 進料分流右昇降  上昇
      OUT     B248  ; 分流右側昇降氣缸C5上昇SV
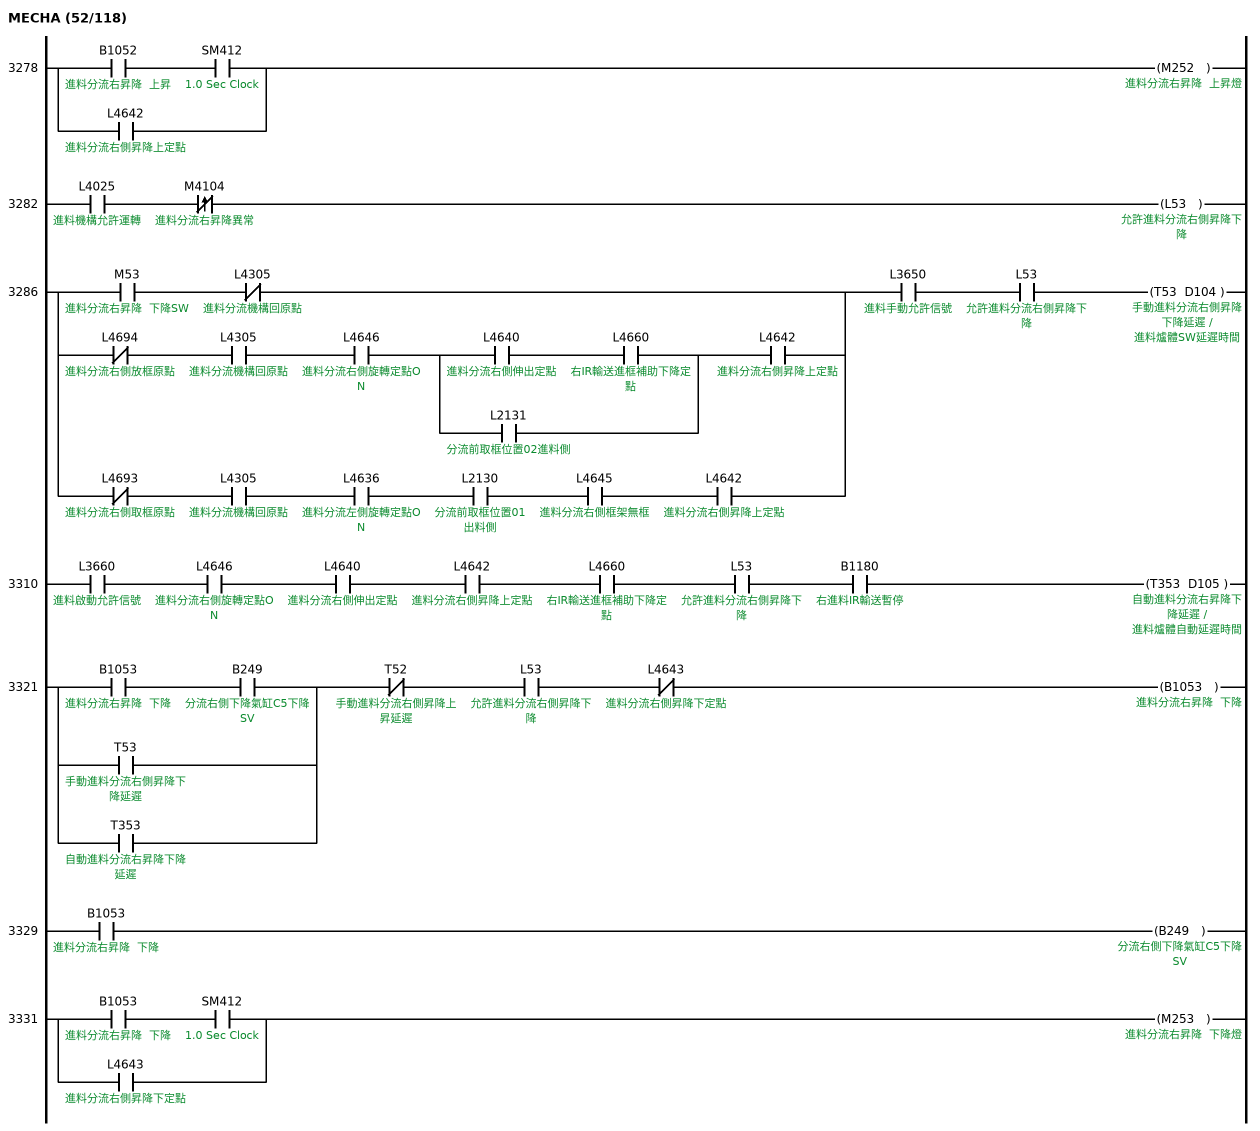
3278  LD      B1052  ; 進料分流右昇降  上昇
      AND     SM412  ; 1.0 Sec Clock
      OR      L4642  ; 進料分流右側昇降上定點
      OUT     M252  ; 進料分流右昇降  上昇燈
3282  LD      L4025  ; 進料機構允許運轉
      ANDPI   M4104  ; 進料分流右昇降異常
      OUT     L53  ; 允許進料分流右側昇降下降
3286  LD      M53  ; 進料分流右昇降  下降SW
      ANI     L4305  ; 進料分流機構回原點
      LDI     L4694  ; 進料分流右側放框原點
      AND     L4305  ; 進料分流機構回原點
      AND     L4646  ; 進料分流右側旋轉定點ON
      LD      L4640  ; 進料分流右側伸出定點
      AND     L4660  ; 右IR輸送進框補助下降定點
      OR      L2131  ; 分流前取框位置02進料側
      ANB
      AND     L4642  ; 進料分流右側昇降上定點
      ORB
      LDI     L4693  ; 進料分流右側取框原點
      AND     L4305  ; 進料分流機構回原點
      AND     L4636  ; 進料分流左側旋轉定點ON
      AND     L2130  ; 分流前取框位置01  出料側
      AND     L4645  ; 進料分流右側框架無框
      AND     L4642  ; 進料分流右側昇降上定點
      ORB
      AND     L3650  ; 進料手動允許信號
      AND     L53  ; 允許進料分流右側昇降下降
      OUT     T53 D104  ; 手動進料分流右側昇降下降延遲 / 進料爐體SW延遲時間
3310  LD      L3660  ; 進料啟動允許信號
      AND     L4646  ; 進料分流右側旋轉定點ON
      AND     L4640  ; 進料分流右側伸出定點
      AND     L4642  ; 進料分流右側昇降上定點
      AND     L4660  ; 右IR輸送進框補助下降定點
      AND     L53  ; 允許進料分流右側昇降下降
      AND     B1180  ; 右進料IR輸送暫停
      OUT     T353 D105  ; 自動進料分流右昇降下降延遲 / 進料爐體自動延遲時間
3321  LD      B1053  ; 進料分流右昇降  下降
      AND     B249  ; 分流右側下降氣缸C5下降SV
      OR      T53  ; 手動進料分流右側昇降下降延遲
      OR      T353  ; 自動進料分流右昇降下降延遲
      ANI     T52  ; 手動進料分流右側昇降上昇延遲
      AND     L53  ; 允許進料分流右側昇降下降
      ANI     L4643  ; 進料分流右側昇降下定點
      OUT     B1053  ; 進料分流右昇降  下降
3329  LD      B1053  ; 進料分流右昇降  下降
      OUT     B249  ; 分流右側下降氣缸C5下降SV
3331  LD      B1053  ; 進料分流右昇降  下降
      AND     SM412  ; 1.0 Sec Clock
      OR      L4643  ; 進料分流右側昇降下定點
      OUT     M253  ; 進料分流右昇降  下降燈
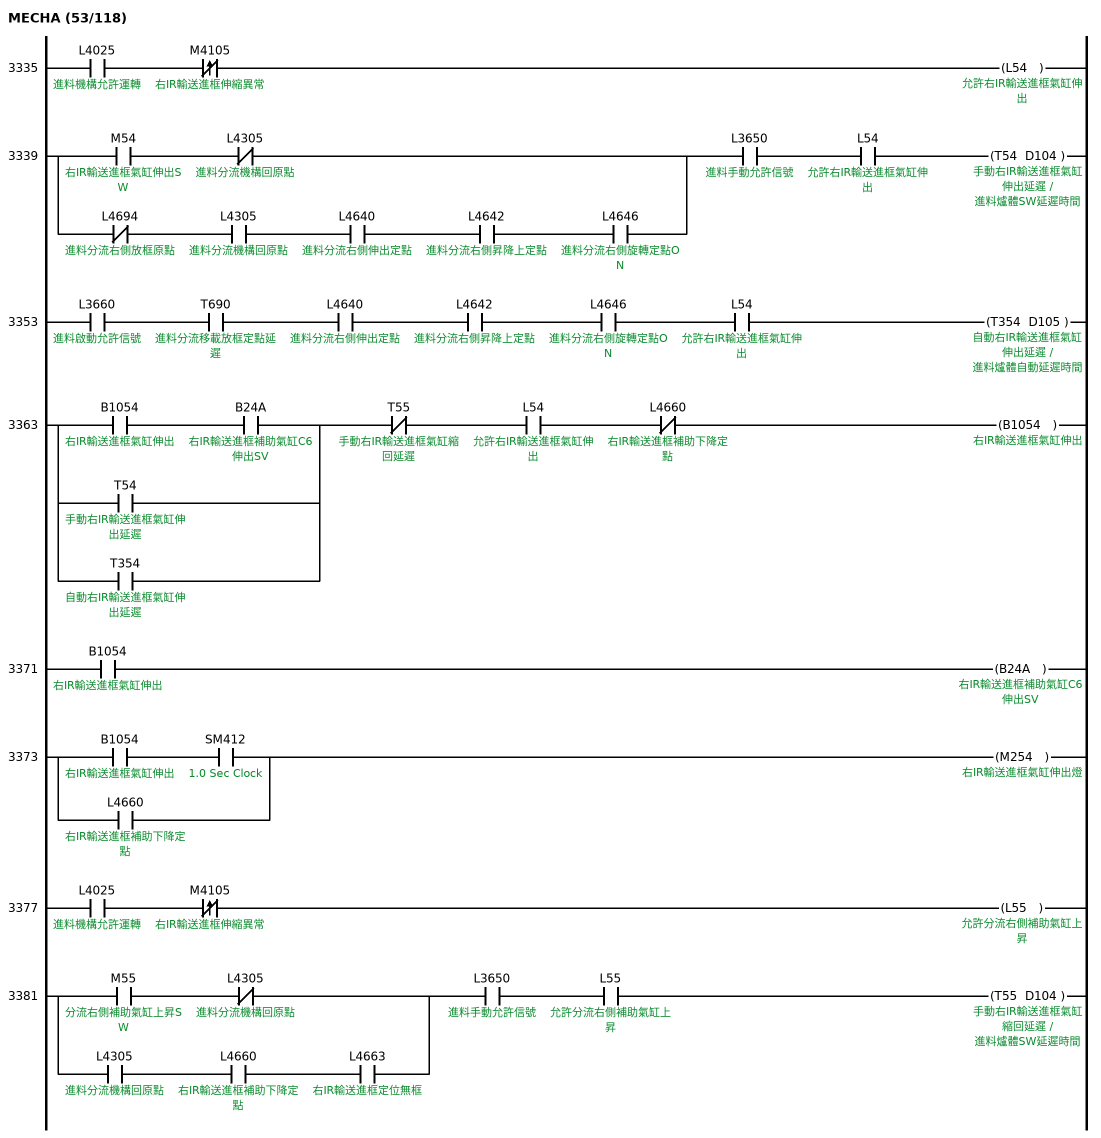
3335  LD      L4025  ; 進料機構允許運轉
      ANDPI   M4105  ; 右IR輸送進框伸縮異常
      OUT     L54  ; 允許右IR輸送進框氣缸伸出
3339  LD      M54  ; 右IR輸送進框氣缸伸出SW
      ANI     L4305  ; 進料分流機構回原點
      LDI     L4694  ; 進料分流右側放框原點
      AND     L4305  ; 進料分流機構回原點
      AND     L4640  ; 進料分流右側伸出定點
      AND     L4642  ; 進料分流右側昇降上定點
      AND     L4646  ; 進料分流右側旋轉定點ON
      ORB
      AND     L3650  ; 進料手動允許信號
      AND     L54  ; 允許右IR輸送進框氣缸伸出
      OUT     T54 D104  ; 手動右IR輸送進框氣缸伸出延遲 / 進料爐體SW延遲時間
3353  LD      L3660  ; 進料啟動允許信號
      AND     T690  ; 進料分流移載放框定點延遲
      AND     L4640  ; 進料分流右側伸出定點
      AND     L4642  ; 進料分流右側昇降上定點
      AND     L4646  ; 進料分流右側旋轉定點ON
      AND     L54  ; 允許右IR輸送進框氣缸伸出
      OUT     T354 D105  ; 自動右IR輸送進框氣缸伸出延遲 / 進料爐體自動延遲時間
3363  LD      B1054  ; 右IR輸送進框氣缸伸出
      AND     B24A  ; 右IR輸送進框補助氣缸C6伸出SV
      OR      T54  ; 手動右IR輸送進框氣缸伸出延遲
      OR      T354  ; 自動右IR輸送進框氣缸伸出延遲
      ANI     T55  ; 手動右IR輸送進框氣缸縮回延遲
      AND     L54  ; 允許右IR輸送進框氣缸伸出
      ANI     L4660  ; 右IR輸送進框補助下降定點
      OUT     B1054  ; 右IR輸送進框氣缸伸出
3371  LD      B1054  ; 右IR輸送進框氣缸伸出
      OUT     B24A  ; 右IR輸送進框補助氣缸C6伸出SV
3373  LD      B1054  ; 右IR輸送進框氣缸伸出
      AND     SM412  ; 1.0 Sec Clock
      OR      L4660  ; 右IR輸送進框補助下降定點
      OUT     M254  ; 右IR輸送進框氣缸伸出燈
3377  LD      L4025  ; 進料機構允許運轉
      ANDPI   M4105  ; 右IR輸送進框伸縮異常
      OUT     L55  ; 允許分流右側補助氣缸上昇
3381  LD      M55  ; 分流右側補助氣缸上昇SW
      ANI     L4305  ; 進料分流機構回原點
      LD      L4305  ; 進料分流機構回原點
      AND     L4660  ; 右IR輸送進框補助下降定點
      AND     L4663  ; 右IR輸送進框定位無框
      ORB
      AND     L3650  ; 進料手動允許信號
      AND     L55  ; 允許分流右側補助氣缸上昇
      OUT     T55 D104  ; 手動右IR輸送進框氣缸縮回延遲 / 進料爐體SW延遲時間
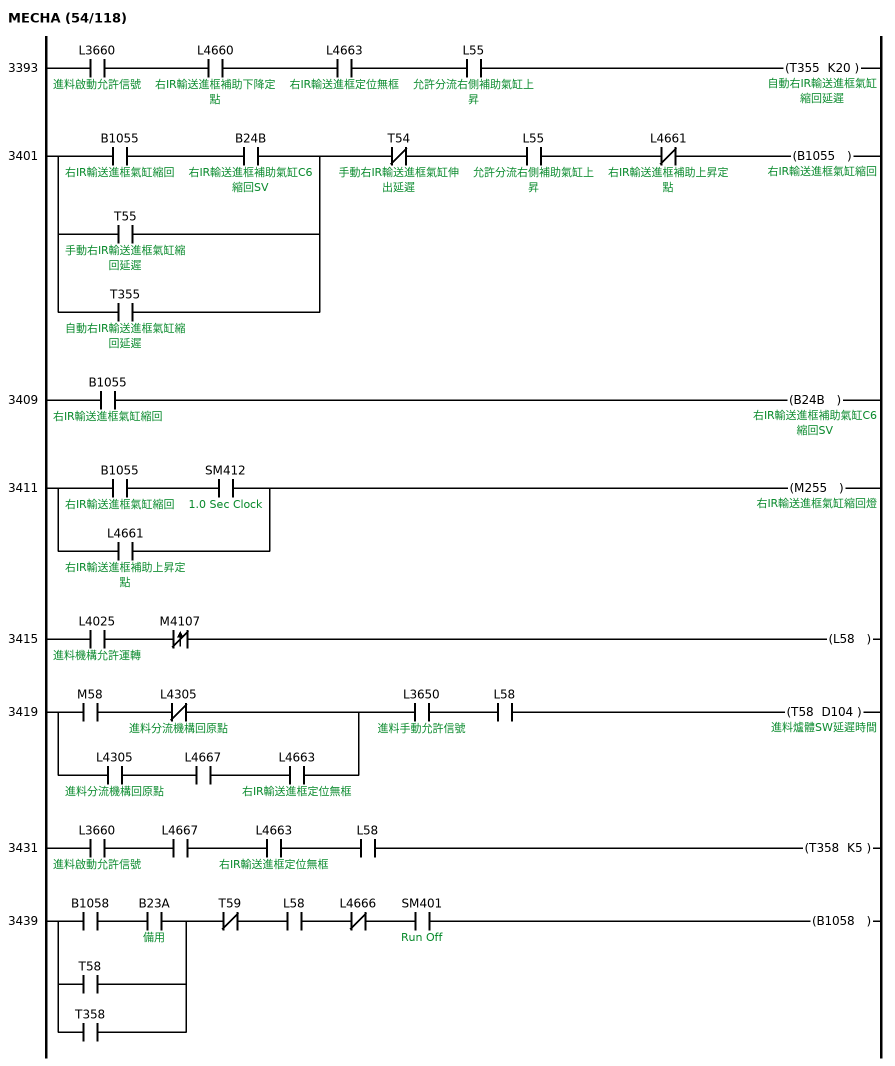
3393  LD      L3660  ; 進料啟動允許信號
      AND     L4660  ; 右IR輸送進框補助下降定點
      AND     L4663  ; 右IR輸送進框定位無框
      AND     L55  ; 允許分流右側補助氣缸上昇
      OUT     T355 K20  ; 自動右IR輸送進框氣缸縮回延遲
3401  LD      B1055  ; 右IR輸送進框氣缸縮回
      AND     B24B  ; 右IR輸送進框補助氣缸C6縮回SV
      OR      T55  ; 手動右IR輸送進框氣缸縮回延遲
      OR      T355  ; 自動右IR輸送進框氣缸縮回延遲
      ANI     T54  ; 手動右IR輸送進框氣缸伸出延遲
      AND     L55  ; 允許分流右側補助氣缸上昇
      ANI     L4661  ; 右IR輸送進框補助上昇定點
      OUT     B1055  ; 右IR輸送進框氣缸縮回
3409  LD      B1055  ; 右IR輸送進框氣缸縮回
      OUT     B24B  ; 右IR輸送進框補助氣缸C6縮回SV
3411  LD      B1055  ; 右IR輸送進框氣缸縮回
      AND     SM412  ; 1.0 Sec Clock
      OR      L4661  ; 右IR輸送進框補助上昇定點
      OUT     M255  ; 右IR輸送進框氣缸縮回燈
3415  LD      L4025  ; 進料機構允許運轉
      ANDPI   M4107
      OUT     L58
3419  LD      M58
      ANI     L4305  ; 進料分流機構回原點
      LD      L4305  ; 進料分流機構回原點
      AND     L4667
      AND     L4663  ; 右IR輸送進框定位無框
      ORB
      AND     L3650  ; 進料手動允許信號
      AND     L58
      OUT     T58 D104  ; 進料爐體SW延遲時間
3431  LD      L3660  ; 進料啟動允許信號
      AND     L4667
      AND     L4663  ; 右IR輸送進框定位無框
      AND     L58
      OUT     T358 K5
3439  LD      B1058
      AND     B23A  ; 備用
      OR      T58
      OR      T358
      ANI     T59
      AND     L58
      ANI     L4666
      AND     SM401  ; Run Off
      OUT     B1058
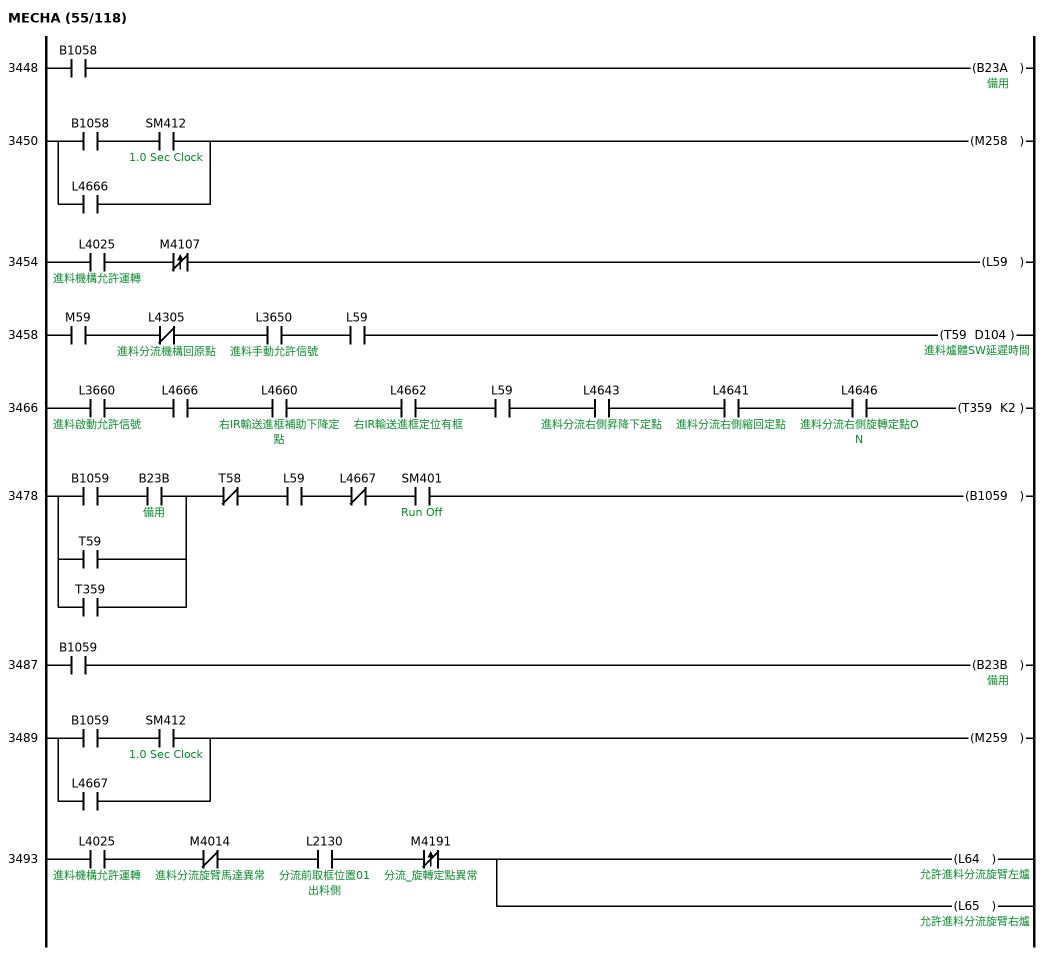
3448  LD      B1058
      OUT     B23A  ; 備用
3450  LD      B1058
      AND     SM412  ; 1.0 Sec Clock
      OR      L4666
      OUT     M258
3454  LD      L4025  ; 進料機構允許運轉
      ANDPI   M4107
      OUT     L59
3458  LD      M59
      ANI     L4305  ; 進料分流機構回原點
      AND     L3650  ; 進料手動允許信號
      AND     L59
      OUT     T59 D104  ; 進料爐體SW延遲時間
3466  LD      L3660  ; 進料啟動允許信號
      AND     L4666
      AND     L4660  ; 右IR輸送進框補助下降定點
      AND     L4662  ; 右IR輸送進框定位有框
      AND     L59
      AND     L4643  ; 進料分流右側昇降下定點
      AND     L4641  ; 進料分流右側縮回定點
      AND     L4646  ; 進料分流右側旋轉定點ON
      OUT     T359 K2
3478  LD      B1059
      AND     B23B  ; 備用
      OR      T59
      OR      T359
      ANI     T58
      AND     L59
      ANI     L4667
      AND     SM401  ; Run Off
      OUT     B1059
3487  LD      B1059
      OUT     B23B  ; 備用
3489  LD      B1059
      AND     SM412  ; 1.0 Sec Clock
      OR      L4667
      OUT     M259
3493  LD      L4025  ; 進料機構允許運轉
      ANI     M4014  ; 進料分流旋臂馬達異常
      AND     L2130  ; 分流前取框位置01  出料側
      ANDPI   M4191  ; 分流_旋轉定點異常
      OUT     L64  ; 允許進料分流旋臂左爐
      OUT     L65  ; 允許進料分流旋臂右爐
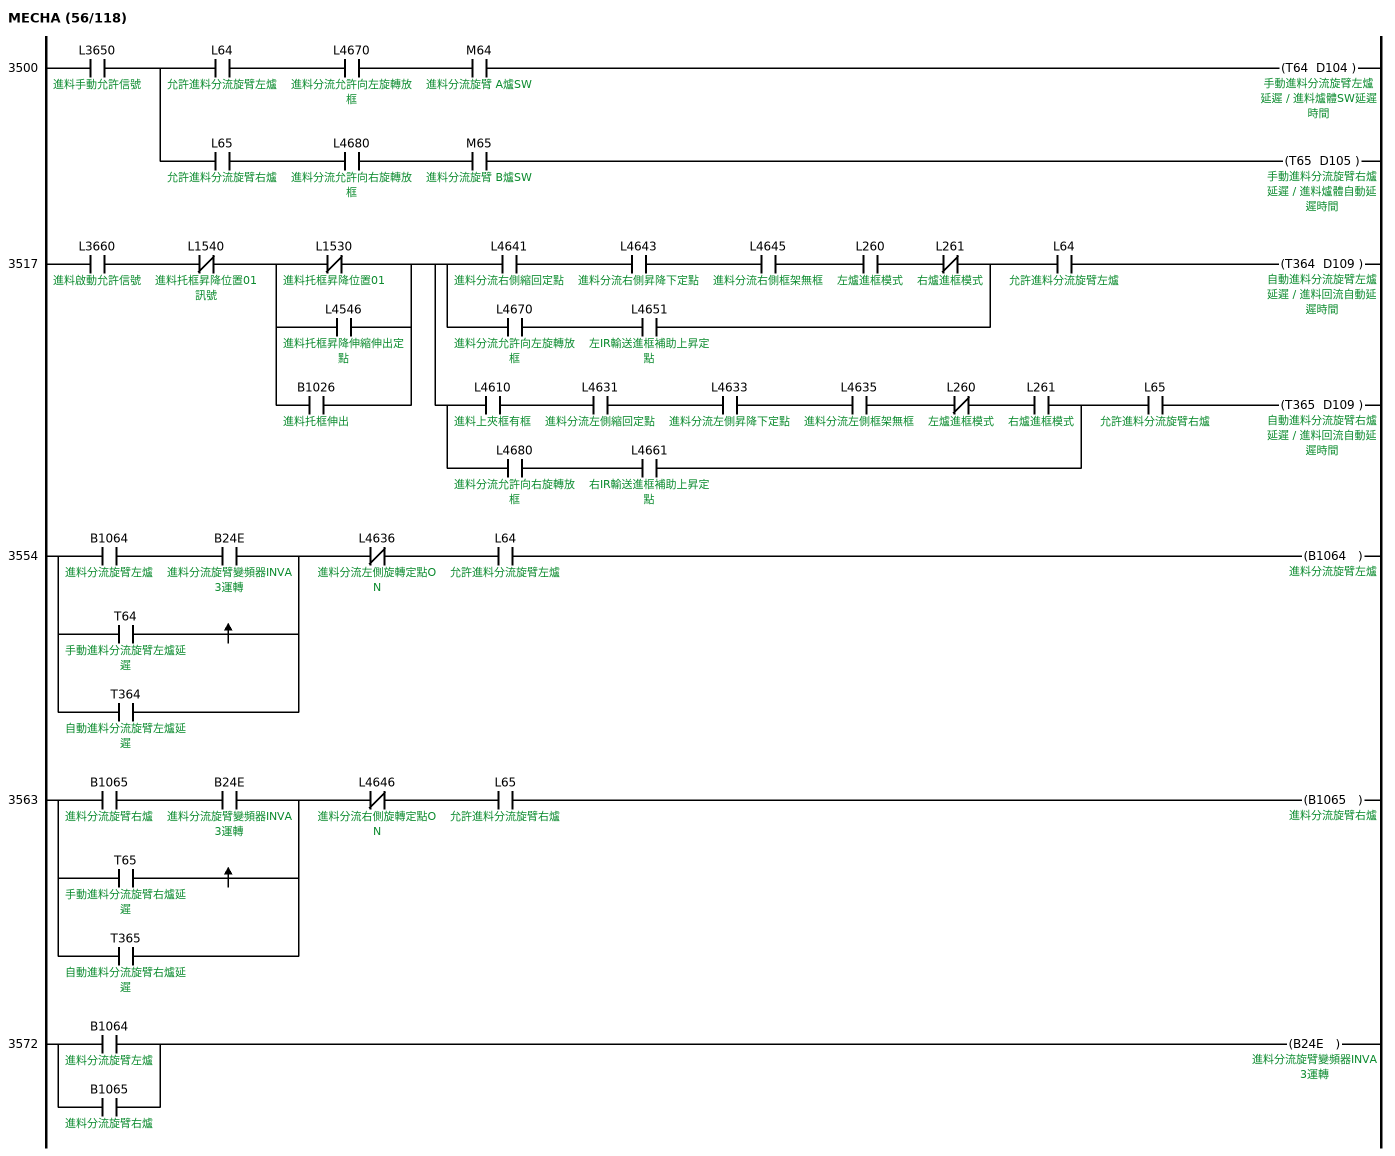
3500  LD      L3650  ; 進料手動允許信號
      MPS
      AND     L64  ; 允許進料分流旋臂左爐
      AND     L4670  ; 進料分流允許向左旋轉放框
      AND     M64  ; 進料分流旋臂 A爐SW
      OUT     T64 D104  ; 手動進料分流旋臂左爐延遲 / 進料爐體SW延遲時間
      MPP
      AND     L65  ; 允許進料分流旋臂右爐
      AND     L4680  ; 進料分流允許向右旋轉放框
      AND     M65  ; 進料分流旋臂 B爐SW
      OUT     T65 D105  ; 手動進料分流旋臂右爐延遲 / 進料爐體自動延遲時間
3517  LD      L3660  ; 進料啟動允許信號
      ANI     L1540  ; 進料托框昇降位置01 訊號
      LDI     L1530  ; 進料托框昇降位置01
      OR      L4546  ; 進料托框昇降伸縮伸出定點
      OR      B1026  ; 進料托框伸出
      ANB
      MPS
      LD      L4641  ; 進料分流右側縮回定點
      AND     L4643  ; 進料分流右側昇降下定點
      AND     L4645  ; 進料分流右側框架無框
      AND     L260  ; 左爐進框模式
      ANI     L261  ; 右爐進框模式
      LD      L4670  ; 進料分流允許向左旋轉放框
      AND     L4651  ; 左IR輸送進框補助上昇定點
      ORB
      ANB
      AND     L64  ; 允許進料分流旋臂左爐
      OUT     T364 D109  ; 自動進料分流旋臂左爐延遲 / 進料回流自動延遲時間
      MPP
      LD      L4610  ; 進料上夾框有框
      AND     L4631  ; 進料分流左側縮回定點
      AND     L4633  ; 進料分流左側昇降下定點
      AND     L4635  ; 進料分流左側框架無框
      ANI     L260  ; 左爐進框模式
      AND     L261  ; 右爐進框模式
      LD      L4680  ; 進料分流允許向右旋轉放框
      AND     L4661  ; 右IR輸送進框補助上昇定點
      ORB
      ANB
      AND     L65  ; 允許進料分流旋臂右爐
      OUT     T365 D109  ; 自動進料分流旋臂右爐延遲 / 進料回流自動延遲時間
3554  LD      B1064  ; 進料分流旋臂左爐
      AND     B24E  ; 進料分流旋臂變頻器INVA3運轉
      LD      T64  ; 手動進料分流旋臂左爐延遲
      MEP
      ORB
      OR      T364  ; 自動進料分流旋臂左爐延遲
      ANI     L4636  ; 進料分流左側旋轉定點ON
      AND     L64  ; 允許進料分流旋臂左爐
      OUT     B1064  ; 進料分流旋臂左爐
3563  LD      B1065  ; 進料分流旋臂右爐
      AND     B24E  ; 進料分流旋臂變頻器INVA3運轉
      LD      T65  ; 手動進料分流旋臂右爐延遲
      MEP
      ORB
      OR      T365  ; 自動進料分流旋臂右爐延遲
      ANI     L4646  ; 進料分流右側旋轉定點ON
      AND     L65  ; 允許進料分流旋臂右爐
      OUT     B1065  ; 進料分流旋臂右爐
3572  LD      B1064  ; 進料分流旋臂左爐
      OR      B1065  ; 進料分流旋臂右爐
      OUT     B24E  ; 進料分流旋臂變頻器INVA3運轉
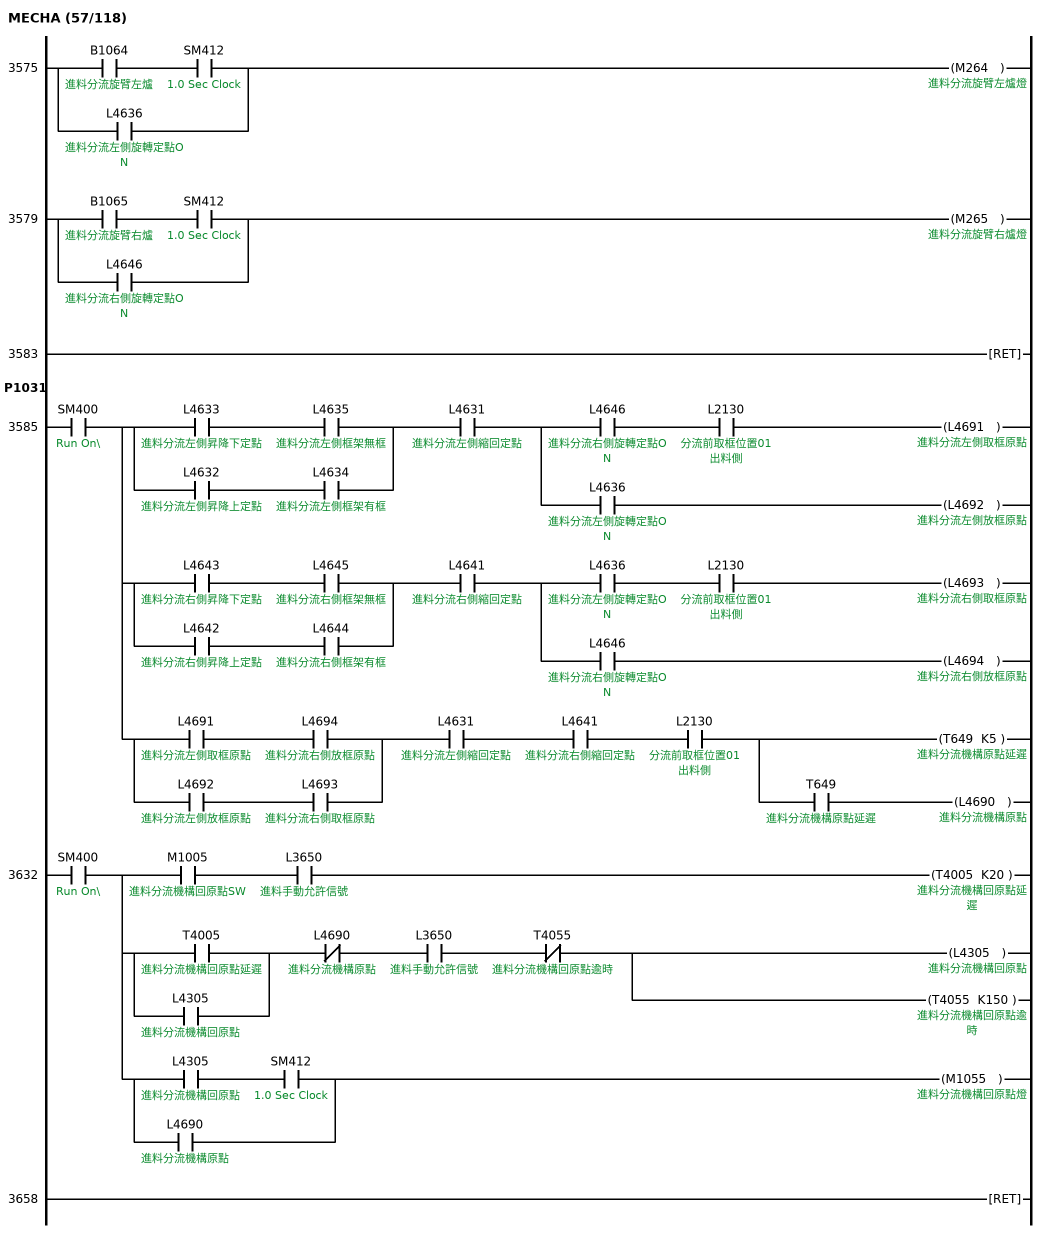
3575  LD      B1064  ; 進料分流旋臂左爐
      AND     SM412  ; 1.0 Sec Clock
      OR      L4636  ; 進料分流左側旋轉定點ON
      OUT     M264  ; 進料分流旋臂左爐燈
3579  LD      B1065  ; 進料分流旋臂右爐
      AND     SM412  ; 1.0 Sec Clock
      OR      L4646  ; 進料分流右側旋轉定點ON
      OUT     M265  ; 進料分流旋臂右爐燈
3583  RET
      P1031
3585  LD      SM400  ; Run On\
      MPS
      LD      L4633  ; 進料分流左側昇降下定點
      AND     L4635  ; 進料分流左側框架無框
      LD      L4632  ; 進料分流左側昇降上定點
      AND     L4634  ; 進料分流左側框架有框
      ORB
      ANB
      AND     L4631  ; 進料分流左側縮回定點
      MPS
      AND     L4646  ; 進料分流右側旋轉定點ON
      AND     L2130  ; 分流前取框位置01  出料側
      OUT     L4691  ; 進料分流左側取框原點
      MPP
      AND     L4636  ; 進料分流左側旋轉定點ON
      OUT     L4692  ; 進料分流左側放框原點
      MRD
      LD      L4643  ; 進料分流右側昇降下定點
      AND     L4645  ; 進料分流右側框架無框
      LD      L4642  ; 進料分流右側昇降上定點
      AND     L4644  ; 進料分流右側框架有框
      ORB
      ANB
      AND     L4641  ; 進料分流右側縮回定點
      MPS
      AND     L4636  ; 進料分流左側旋轉定點ON
      AND     L2130  ; 分流前取框位置01  出料側
      OUT     L4693  ; 進料分流右側取框原點
      MPP
      AND     L4646  ; 進料分流右側旋轉定點ON
      OUT     L4694  ; 進料分流右側放框原點
      MPP
      LD      L4691  ; 進料分流左側取框原點
      AND     L4694  ; 進料分流右側放框原點
      LD      L4692  ; 進料分流左側放框原點
      AND     L4693  ; 進料分流右側取框原點
      ORB
      ANB
      AND     L4631  ; 進料分流左側縮回定點
      AND     L4641  ; 進料分流右側縮回定點
      AND     L2130  ; 分流前取框位置01  出料側
      OUT     T649 K5  ; 進料分流機構原點延遲
      AND     T649  ; 進料分流機構原點延遲
      OUT     L4690  ; 進料分流機構原點
3632  LD      SM400  ; Run On\
      MPS
      AND     M1005  ; 進料分流機構回原點SW
      AND     L3650  ; 進料手動允許信號
      OUT     T4005 K20  ; 進料分流機構回原點延遲
      MRD
      LD      T4005  ; 進料分流機構回原點延遲
      OR      L4305  ; 進料分流機構回原點
      ANB
      ANI     L4690  ; 進料分流機構原點
      AND     L3650  ; 進料手動允許信號
      ANI     T4055  ; 進料分流機構回原點逾時
      OUT     L4305  ; 進料分流機構回原點
      OUT     T4055 K150  ; 進料分流機構回原點逾時
      MPP
      LD      L4305  ; 進料分流機構回原點
      AND     SM412  ; 1.0 Sec Clock
      OR      L4690  ; 進料分流機構原點
      ANB
      OUT     M1055  ; 進料分流機構回原點燈
3658  RET
; ---------回流輸送---------
      P1012
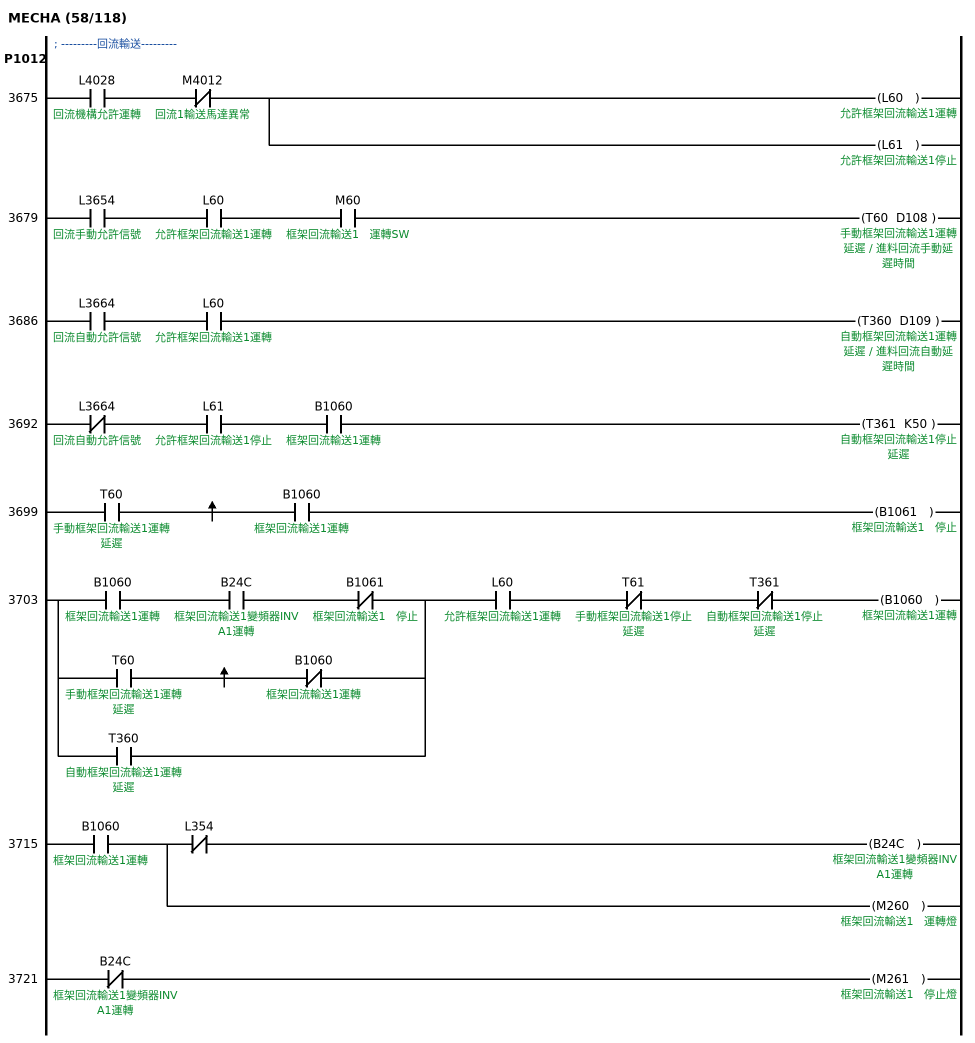
3675  LD      L4028  ; 回流機構允許運轉
      ANI     M4012  ; 回流1輸送馬達異常
      OUT     L60  ; 允許框架回流輸送1運轉
      OUT     L61  ; 允許框架回流輸送1停止
3679  LD      L3654  ; 回流手動允許信號
      AND     L60  ; 允許框架回流輸送1運轉
      AND     M60  ; 框架回流輸送1   運轉SW
      OUT     T60 D108  ; 手動框架回流輸送1運轉延遲 / 進料回流手動延遲時間
3686  LD      L3664  ; 回流自動允許信號
      AND     L60  ; 允許框架回流輸送1運轉
      OUT     T360 D109  ; 自動框架回流輸送1運轉延遲 / 進料回流自動延遲時間
3692  LDI     L3664  ; 回流自動允許信號
      AND     L61  ; 允許框架回流輸送1停止
      AND     B1060  ; 框架回流輸送1運轉
      OUT     T361 K50  ; 自動框架回流輸送1停止延遲
3699  LD      T60  ; 手動框架回流輸送1運轉延遲
      MEP
      AND     B1060  ; 框架回流輸送1運轉
      OUT     B1061  ; 框架回流輸送1   停止
3703  LD      B1060  ; 框架回流輸送1運轉
      AND     B24C  ; 框架回流輸送1變頻器INVA1運轉
      ANI     B1061  ; 框架回流輸送1   停止
      LD      T60  ; 手動框架回流輸送1運轉延遲
      MEP
      ANI     B1060  ; 框架回流輸送1運轉
      ORB
      OR      T360  ; 自動框架回流輸送1運轉延遲
      AND     L60  ; 允許框架回流輸送1運轉
      ANI     T61  ; 手動框架回流輸送1停止延遲
      ANI     T361  ; 自動框架回流輸送1停止延遲
      OUT     B1060  ; 框架回流輸送1運轉
3715  LD      B1060  ; 框架回流輸送1運轉
      MPS
      ANI     L354
      OUT     B24C  ; 框架回流輸送1變頻器INVA1運轉
      MPP
      OUT     M260  ; 框架回流輸送1   運轉燈
3721  LDI     B24C  ; 框架回流輸送1變頻器INVA1運轉
      OUT     M261  ; 框架回流輸送1   停止燈
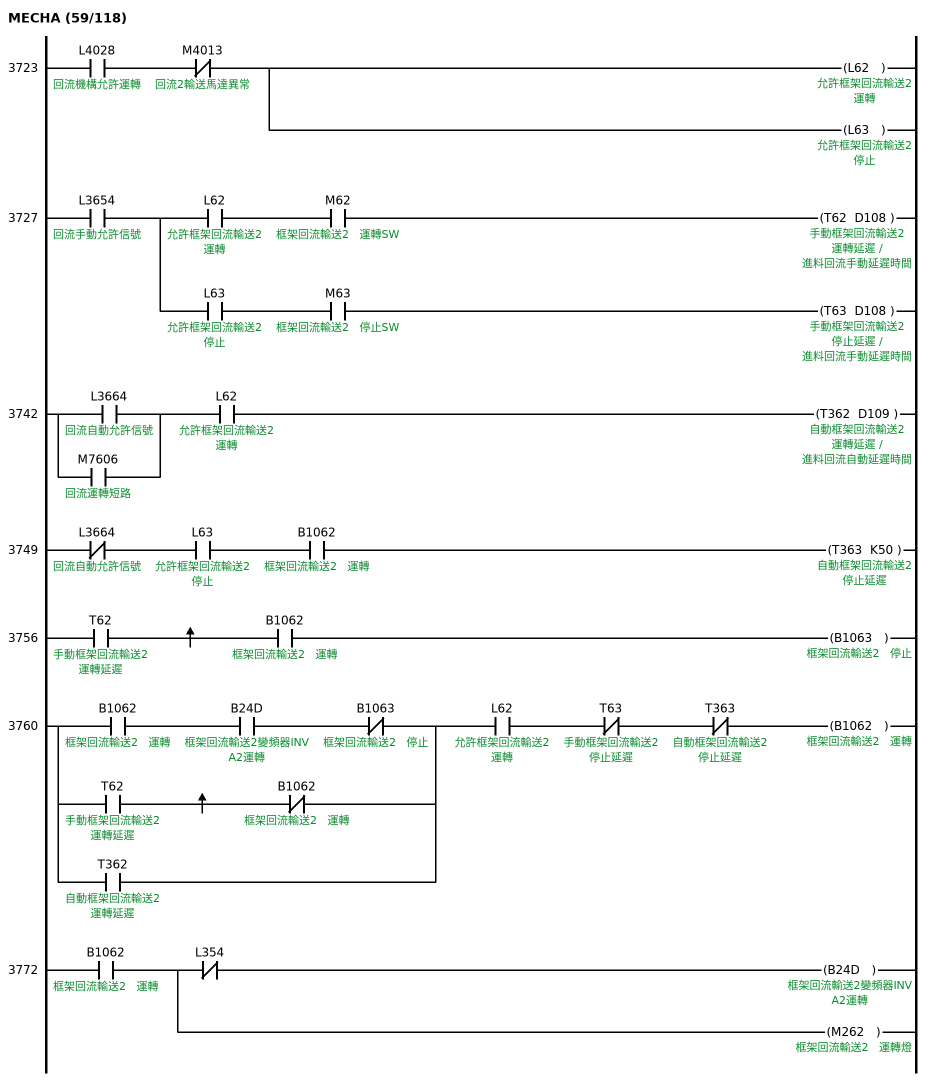
3723  LD      L4028  ; 回流機構允許運轉
      ANI     M4013  ; 回流2輸送馬達異常
      OUT     L62  ; 允許框架回流輸送2   運轉
      OUT     L63  ; 允許框架回流輸送2   停止
3727  LD      L3654  ; 回流手動允許信號
      MPS
      AND     L62  ; 允許框架回流輸送2   運轉
      AND     M62  ; 框架回流輸送2   運轉SW
      OUT     T62 D108  ; 手動框架回流輸送2   運轉延遲 / 進料回流手動延遲時間
      MPP
      AND     L63  ; 允許框架回流輸送2   停止
      AND     M63  ; 框架回流輸送2   停止SW
      OUT     T63 D108  ; 手動框架回流輸送2   停止延遲 / 進料回流手動延遲時間
3742  LD      L3664  ; 回流自動允許信號
      OR      M7606  ; 回流運轉短路
      AND     L62  ; 允許框架回流輸送2   運轉
      OUT     T362 D109  ; 自動框架回流輸送2   運轉延遲 / 進料回流自動延遲時間
3749  LDI     L3664  ; 回流自動允許信號
      AND     L63  ; 允許框架回流輸送2   停止
      AND     B1062  ; 框架回流輸送2   運轉
      OUT     T363 K50  ; 自動框架回流輸送2   停止延遲
3756  LD      T62  ; 手動框架回流輸送2   運轉延遲
      MEP
      AND     B1062  ; 框架回流輸送2   運轉
      OUT     B1063  ; 框架回流輸送2   停止
3760  LD      B1062  ; 框架回流輸送2   運轉
      AND     B24D  ; 框架回流輸送2變頻器INVA2運轉
      ANI     B1063  ; 框架回流輸送2   停止
      LD      T62  ; 手動框架回流輸送2   運轉延遲
      MEP
      ANI     B1062  ; 框架回流輸送2   運轉
      ORB
      OR      T362  ; 自動框架回流輸送2   運轉延遲
      AND     L62  ; 允許框架回流輸送2   運轉
      ANI     T63  ; 手動框架回流輸送2   停止延遲
      ANI     T363  ; 自動框架回流輸送2   停止延遲
      OUT     B1062  ; 框架回流輸送2   運轉
3772  LD      B1062  ; 框架回流輸送2   運轉
      MPS
      ANI     L354
      OUT     B24D  ; 框架回流輸送2變頻器INVA2運轉
      MPP
      OUT     M262  ; 框架回流輸送2   運轉燈
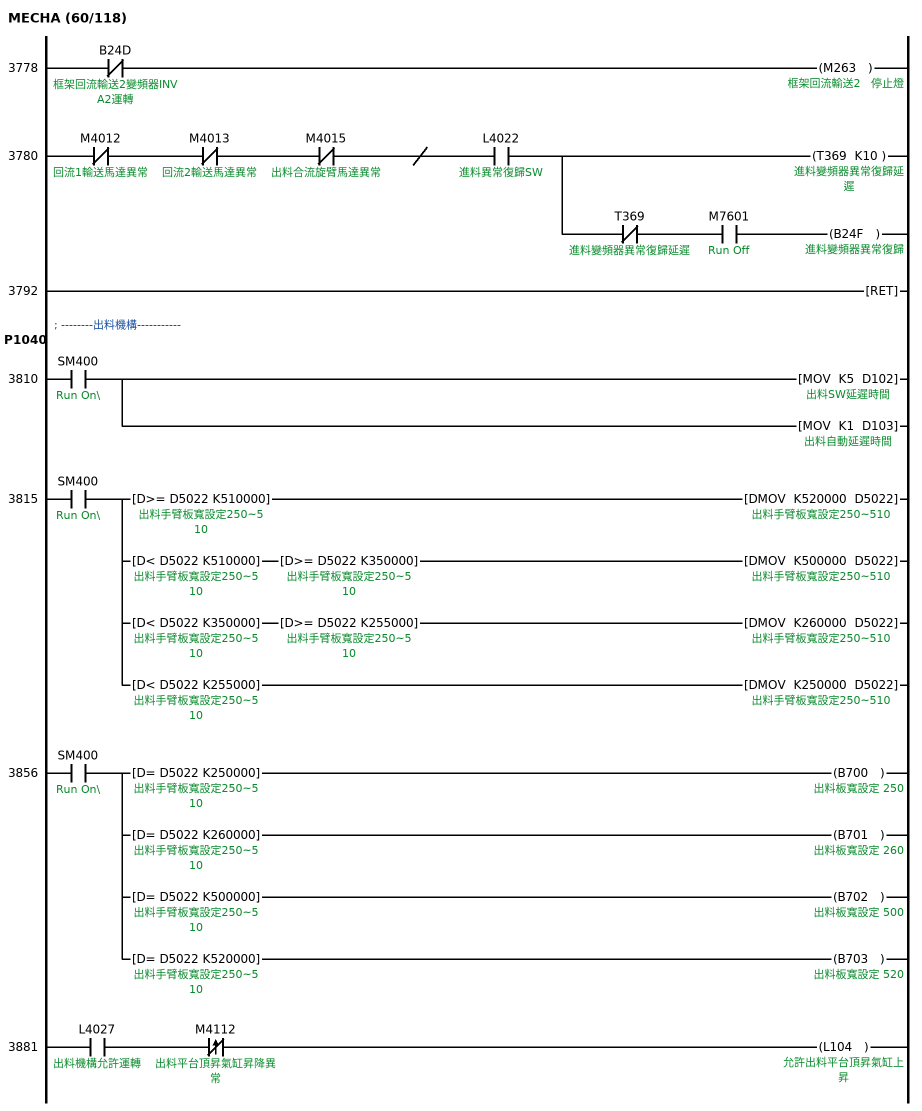
3778  LDI     B24D  ; 框架回流輸送2變頻器INVA2運轉
      OUT     M263  ; 框架回流輸送2   停止燈
3780  LDI     M4012  ; 回流1輸送馬達異常
      ANI     M4013  ; 回流2輸送馬達異常
      ANI     M4015  ; 出料合流旋臂馬達異常
      INV
      AND     L4022  ; 進料異常復歸SW
      OUT     T369 K10  ; 進料變頻器異常復歸延遲
      ANI     T369  ; 進料變頻器異常復歸延遲
      AND     M7601  ; Run Off
      OUT     B24F  ; 進料變頻器異常復歸
3792  RET
; --------出料機構-----------
      P1040
3810  LD      SM400  ; Run On\
      MOV     K5 D102  ; 出料SW延遲時間
      MOV     K1 D103  ; 出料自動延遲時間
3815  LD      SM400  ; Run On\
      MPS
      ANDD>=  D5022 K510000  ; 出料手臂板寬設定250~510
      DMOV    K520000 D5022
      MRD
      ANDD<   D5022 K510000  ; 出料手臂板寬設定250~510
      ANDD>=  D5022 K350000  ; 出料手臂板寬設定250~510
      DMOV    K500000 D5022
      MRD
      ANDD<   D5022 K350000  ; 出料手臂板寬設定250~510
      ANDD>=  D5022 K255000  ; 出料手臂板寬設定250~510
      DMOV    K260000 D5022
      MPP
      ANDD<   D5022 K255000  ; 出料手臂板寬設定250~510
      DMOV    K250000 D5022
3856  LD      SM400  ; Run On\
      MPS
      ANDD=   D5022 K250000  ; 出料手臂板寬設定250~510
      OUT     B700  ; 出料板寬設定 250
      MRD
      ANDD=   D5022 K260000  ; 出料手臂板寬設定250~510
      OUT     B701  ; 出料板寬設定 260
      MRD
      ANDD=   D5022 K500000  ; 出料手臂板寬設定250~510
      OUT     B702  ; 出料板寬設定 500
      MPP
      ANDD=   D5022 K520000  ; 出料手臂板寬設定250~510
      OUT     B703  ; 出料板寬設定 520
3881  LD      L4027  ; 出料機構允許運轉
      ANDPI   M4112  ; 出料平台頂昇氣缸昇降異常
      OUT     L104  ; 允許出料平台頂昇氣缸上昇
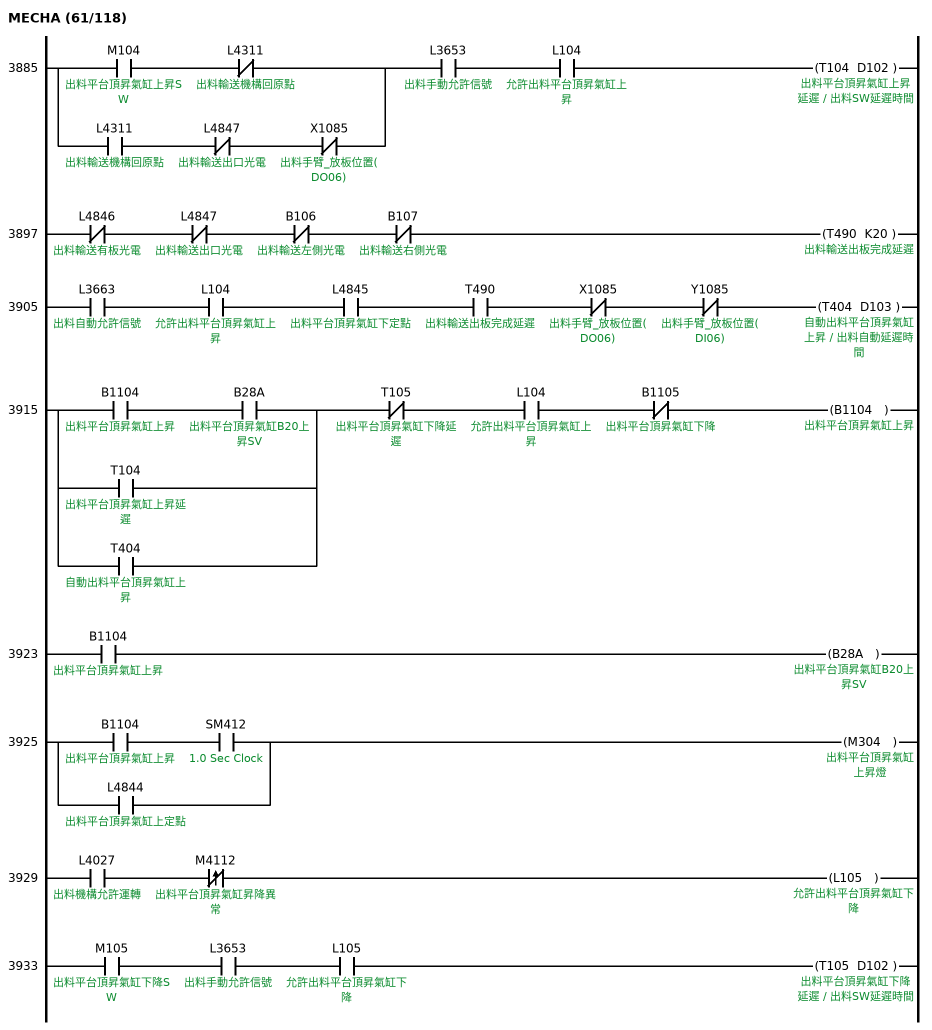
3885  LD      M104  ; 出料平台頂昇氣缸上昇SW
      ANI     L4311  ; 出料輸送機構回原點
      LD      L4311  ; 出料輸送機構回原點
      ANI     L4847  ; 出料輸送出口光電
      ANI     X1085  ; 出料手臂_放板位置(DO06)
      ORB
      AND     L3653  ; 出料手動允許信號
      AND     L104  ; 允許出料平台頂昇氣缸上昇
      OUT     T104 D102  ; 出料平台頂昇氣缸上昇延遲 / 出料SW延遲時間
3897  LDI     L4846  ; 出料輸送有板光電
      ANI     L4847  ; 出料輸送出口光電
      ANI     B106  ; 出料輸送左側光電
      ANI     B107  ; 出料輸送右側光電
      OUT     T490 K20  ; 出料輸送出板完成延遲
3905  LD      L3663  ; 出料自動允許信號
      AND     L104  ; 允許出料平台頂昇氣缸上昇
      AND     L4845  ; 出料平台頂昇氣缸下定點
      AND     T490  ; 出料輸送出板完成延遲
      ANI     X1085  ; 出料手臂_放板位置(DO06)
      ANI     Y1085  ; 出料手臂_放板位置(DI06)
      OUT     T404 D103  ; 自動出料平台頂昇氣缸上昇 / 出料自動延遲時間
3915  LD      B1104  ; 出料平台頂昇氣缸上昇
      AND     B28A  ; 出料平台頂昇氣缸B20上昇SV
      OR      T104  ; 出料平台頂昇氣缸上昇延遲
      OR      T404  ; 自動出料平台頂昇氣缸上昇
      ANI     T105  ; 出料平台頂昇氣缸下降延遲
      AND     L104  ; 允許出料平台頂昇氣缸上昇
      ANI     B1105  ; 出料平台頂昇氣缸下降
      OUT     B1104  ; 出料平台頂昇氣缸上昇
3923  LD      B1104  ; 出料平台頂昇氣缸上昇
      OUT     B28A  ; 出料平台頂昇氣缸B20上昇SV
3925  LD      B1104  ; 出料平台頂昇氣缸上昇
      AND     SM412  ; 1.0 Sec Clock
      OR      L4844  ; 出料平台頂昇氣缸上定點
      OUT     M304  ; 出料平台頂昇氣缸  上昇燈
3929  LD      L4027  ; 出料機構允許運轉
      ANDPI   M4112  ; 出料平台頂昇氣缸昇降異常
      OUT     L105  ; 允許出料平台頂昇氣缸下降
3933  LD      M105  ; 出料平台頂昇氣缸下降SW
      AND     L3653  ; 出料手動允許信號
      AND     L105  ; 允許出料平台頂昇氣缸下降
      OUT     T105 D102  ; 出料平台頂昇氣缸下降延遲 / 出料SW延遲時間
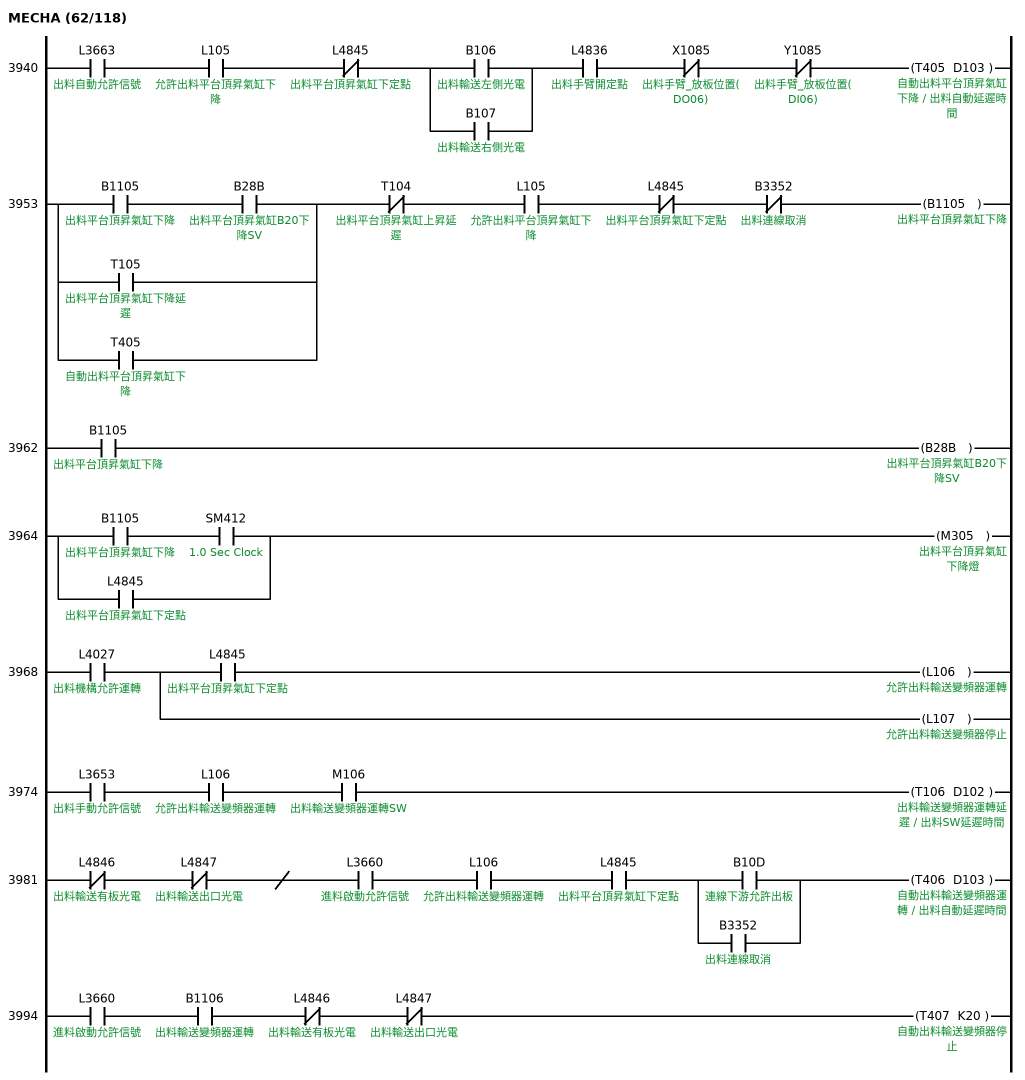
3940  LD      L3663  ; 出料自動允許信號
      AND     L105  ; 允許出料平台頂昇氣缸下降
      ANI     L4845  ; 出料平台頂昇氣缸下定點
      LD      B106  ; 出料輸送左側光電
      OR      B107  ; 出料輸送右側光電
      ANB
      AND     L4836  ; 出料手臂開定點
      ANI     X1085  ; 出料手臂_放板位置(DO06)
      ANI     Y1085  ; 出料手臂_放板位置(DI06)
      OUT     T405 D103  ; 自動出料平台頂昇氣缸下降 / 出料自動延遲時間
3953  LD      B1105  ; 出料平台頂昇氣缸下降
      AND     B28B  ; 出料平台頂昇氣缸B20下降SV
      OR      T105  ; 出料平台頂昇氣缸下降延遲
      OR      T405  ; 自動出料平台頂昇氣缸下降
      ANI     T104  ; 出料平台頂昇氣缸上昇延遲
      AND     L105  ; 允許出料平台頂昇氣缸下降
      ANI     L4845  ; 出料平台頂昇氣缸下定點
      ANI     B3352  ; 出料連線取消
      OUT     B1105  ; 出料平台頂昇氣缸下降
3962  LD      B1105  ; 出料平台頂昇氣缸下降
      OUT     B28B  ; 出料平台頂昇氣缸B20下降SV
3964  LD      B1105  ; 出料平台頂昇氣缸下降
      AND     SM412  ; 1.0 Sec Clock
      OR      L4845  ; 出料平台頂昇氣缸下定點
      OUT     M305  ; 出料平台頂昇氣缸  下降燈
3968  LD      L4027  ; 出料機構允許運轉
      MPS
      AND     L4845  ; 出料平台頂昇氣缸下定點
      OUT     L106  ; 允許出料輸送變頻器運轉
      MPP
      OUT     L107  ; 允許出料輸送變頻器停止
3974  LD      L3653  ; 出料手動允許信號
      AND     L106  ; 允許出料輸送變頻器運轉
      AND     M106  ; 出料輸送變頻器運轉SW
      OUT     T106 D102  ; 出料輸送變頻器運轉延遲 / 出料SW延遲時間
3981  LDI     L4846  ; 出料輸送有板光電
      ANI     L4847  ; 出料輸送出口光電
      INV
      AND     L3660  ; 進料啟動允許信號
      AND     L106  ; 允許出料輸送變頻器運轉
      AND     L4845  ; 出料平台頂昇氣缸下定點
      LD      B10D  ; 連線下游允許出板
      OR      B3352  ; 出料連線取消
      ANB
      OUT     T406 D103  ; 自動出料輸送變頻器運轉 / 出料自動延遲時間
3994  LD      L3660  ; 進料啟動允許信號
      AND     B1106  ; 出料輸送變頻器運轉
      ANI     L4846  ; 出料輸送有板光電
      ANI     L4847  ; 出料輸送出口光電
      OUT     T407 K20  ; 自動出料輸送變頻器停止
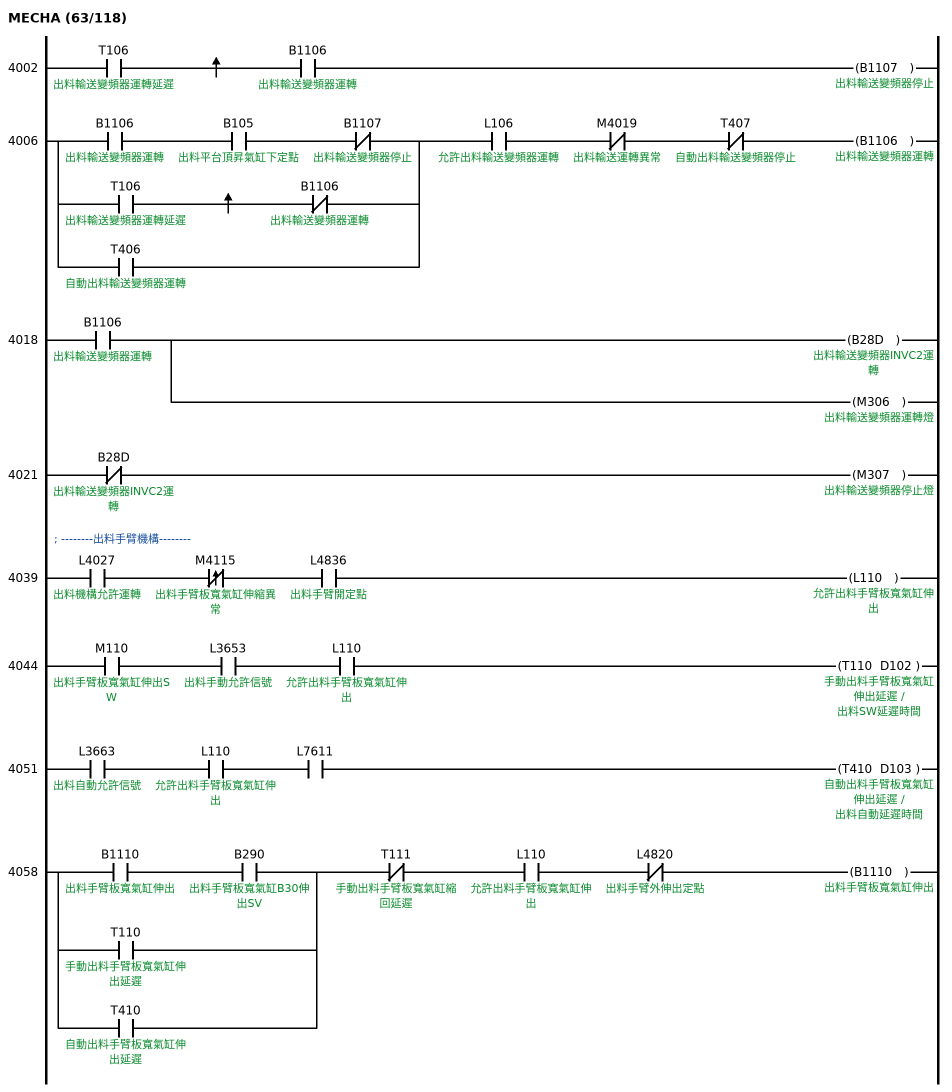
4002  LD      T106  ; 出料輸送變頻器運轉延遲
      MEP
      AND     B1106  ; 出料輸送變頻器運轉
      OUT     B1107  ; 出料輸送變頻器停止
4006  LD      B1106  ; 出料輸送變頻器運轉
      AND     B105  ; 出料平台頂昇氣缸下定點
      ANI     B1107  ; 出料輸送變頻器停止
      LD      T106  ; 出料輸送變頻器運轉延遲
      MEP
      ANI     B1106  ; 出料輸送變頻器運轉
      ORB
      OR      T406  ; 自動出料輸送變頻器運轉
      AND     L106  ; 允許出料輸送變頻器運轉
      ANI     M4019  ; 出料輸送運轉異常
      ANI     T407  ; 自動出料輸送變頻器停止
      OUT     B1106  ; 出料輸送變頻器運轉
4018  LD      B1106  ; 出料輸送變頻器運轉
      OUT     B28D  ; 出料輸送變頻器INVC2運轉
      OUT     M306  ; 出料輸送變頻器運轉燈
4021  LDI     B28D  ; 出料輸送變頻器INVC2運轉
      OUT     M307  ; 出料輸送變頻器停止燈
; --------出料手臂機構--------
4039  LD      L4027  ; 出料機構允許運轉
      ANDPI   M4115  ; 出料手臂板寬氣缸伸縮異常
      AND     L4836  ; 出料手臂開定點
      OUT     L110  ; 允許出料手臂板寬氣缸伸出
4044  LD      M110  ; 出料手臂板寬氣缸伸出SW
      AND     L3653  ; 出料手動允許信號
      AND     L110  ; 允許出料手臂板寬氣缸伸出
      OUT     T110 D102  ; 手動出料手臂板寬氣缸伸出延遲 / 出料SW延遲時間
4051  LD      L3663  ; 出料自動允許信號
      AND     L110  ; 允許出料手臂板寬氣缸伸出
      AND     L7611
      OUT     T410 D103  ; 自動出料手臂板寬氣缸伸出延遲 / 出料自動延遲時間
4058  LD      B1110  ; 出料手臂板寬氣缸伸出
      AND     B290  ; 出料手臂板寬氣缸B30伸出SV
      OR      T110  ; 手動出料手臂板寬氣缸伸出延遲
      OR      T410  ; 自動出料手臂板寬氣缸伸出延遲
      ANI     T111  ; 手動出料手臂板寬氣缸縮回延遲
      AND     L110  ; 允許出料手臂板寬氣缸伸出
      ANI     L4820  ; 出料手臂外伸出定點
      OUT     B1110  ; 出料手臂板寬氣缸伸出
